LIN {X 0,Y 509.214,Z 871.751,A -85,B 0,C 180,E1 -5495.544,E2 -5495.544} C_VEL
LIN {X 0,Y 509.315,Z 866.896,A -85,B 0,C 180,E1 -5497.532,E2 -5497.532} C_VEL
LIN {X 0,Y 509.382,Z 861.752,A -85,B 0,C 180,E1 -5499.129,E2 -5499.129} C_VEL
LIN {X 0,Y 509.592,Z 855.435,A -85,B 0,C 180,E1 -5500.73,E2 -5500.73} C_VEL
LIN {X 0,Y 509.89,Z 847.858,A -85,B 0,C 180,E1 -5502.336,E2 -5502.336} C_VEL
LIN {X 0,Y 510.189,Z 840.077,A -85,B 0,C 180,E1 -5503.746,E2 -5503.746} C_VEL
LIN {X 0,Y 510.685,Z 831.046,A -85,B 0,C 180,E1 -5505.157,E2 -5505.157} C_VEL
LIN {X 0,Y 511.176,Z 820.613,A -85,B 0,C 180,E1 -5506.575,E2 -5506.575} C_VEL
LIN {X 0,Y 511.842,Z 808.389,A -85,B 0,C 180,E1 -5507.995,E2 -5507.995} C_VEL
LIN {X 0,Y 512.559,Z 796.031,A -85,B 0,C 180,E1 -5509.212,E2 -5509.212} C_VEL
LIN {X 0,Y 513.225,Z 784.136,A -85,B 0,C 180,E1 -5510.228,E2 -5510.228} C_VEL
LIN {X 0,Y 513.912,Z 772.243,A -85,B 0,C 180,E1 -5511.108,E2 -5511.108} C_VEL
LIN {X 0,Y 514.522,Z 760.984,A -85,B 0,C 180,E1 -5511.831,E2 -5511.831} C_VEL
LIN {X 0,Y 515.084,Z 748.665,A -85,B 0,C 180,E1 -5512.513,E2 -5512.513} C_VEL
LIN {X 0,Y 515.68,Z 735.496,A -85,B 0,C 180,E1 -5513.12,E2 -5513.12} C_VEL
LIN {X 0,Y 516.156,Z 722.774,A -85,B 0,C 180,E1 -5513.602,E2 -5513.602} C_VEL
LIN {X 0,Y 516.519,Z 710.205,A -85,B 0,C 180,E1 -5513.984,E2 -5513.984} C_VEL
LIN {X 0,Y 516.865,Z 696.063,A -85,B 0,C 180,E1 -5514.301,E2 -5514.301} C_VEL
LIN {X 0,Y 517.478,Z 641.628,A -85,B 0,C 180,E1 -5515.113,E2 -5515.113} C_VEL
LIN {X 0,Y 518.755,Z 504.01,A -85,B 0,C 180,E1 -5517.123,E2 -5517.123} C_VEL
LIN {X 0,Y 513.714,Z 483.814,A -85,B 0,C 180,E1 -5517.747,E2 -5517.747} C_VEL
LIN {X 0,Y 514.557,Z 463.773,A -85,B 0,C 180,E1 -5520.63,E2 -5520.63} C_VEL
LIN {X 0,Y 513.302,Z 457.477,A -85,B 0,C 180,E1 -5521.652,E2 -5521.652} C_VEL
LIN {X 0,Y 509.894,Z 444.343,A -85,B 0,C 180,E1 -5523.932,E2 -5523.932} C_VEL
LIN {X 0,Y 509.819,Z 444.213,A -85,B 0,C 180,E1 -5526.913,E2 -5526.913} C_VEL
LIN {X 0,Y 509.829,Z 444.217,A -85,B 0,C 180,E1 -5529.47,E2 -5529.47} C_VEL
LIN {X 0,Y 509.828,Z 444.222,A -85,B 0,C 180,E1 -5532.489,E2 -5532.489} C_VEL
LIN {X 0,Y 509.851,Z 444.222,A -85,B 0,C 180,E1 -5535.332,E2 -5535.332} C_VEL
LIN {X 0,Y 509.859,Z 444.219,A -85,B 0,C 180,E1 -5538.575,E2 -5538.575} C_VEL
LIN {X 0,Y 509.846,Z 444.227,A -85,B 0,C 180,E1 -5541.786,E2 -5541.786} C_VEL
LIN {X 0,Y 509.839,Z 444.212,A -85,B 0,C 180,E1 -5544.623,E2 -5544.623} C_VEL
LIN {X 0,Y 509.858,Z 444.222,A -85,B 0,C 180,E1 -5547.481,E2 -5547.481} C_VEL
LIN {X 0,Y 509.873,Z 444.209,A -85,B 0,C 180,E1 -5550.269,E2 -5550.269} C_VEL
LIN {X 0,Y 509.879,Z 444.208,A -85,B 0,C 180,E1 -5552.944,E2 -5552.944} C_VEL
LIN {X 0,Y 509.861,Z 444.222,A -85,B 0,C 180,E1 -5555.574,E2 -5555.574} C_VEL
LIN {X 0,Y 509.842,Z 444.205,A -85,B 0,C 180,E1 -5558.998,E2 -5558.998} C_VEL
LIN {X 0,Y 509.879,Z 444.21,A -85,B 0,C 180,E1 -5561.999,E2 -5561.999} C_VEL
LIN {X 0,Y 509.901,Z 444.215,A -85,B 0,C 180,E1 -5564.818,E2 -5564.818} C_VEL
LIN {X 0,Y 509.896,Z 444.218,A -85,B 0,C 180,E1 -5568.121,E2 -5568.121} C_VEL
LIN {X 0,Y 509.909,Z 444.207,A -85,B 0,C 180,E1 -5571.28,E2 -5571.28} C_VEL
LIN {X 0,Y 509.969,Z 444.207,A -85,B 0,C 180,E1 -5573.67,E2 -5573.67} C_VEL
LIN {X 0,Y 510.046,Z 444.194,A -85,B 0,C 180,E1 -5577.631,E2 -5577.631} C_VEL
LIN {X 0,Y 510.056,Z 444.192,A -85,B 0,C 180,E1 -5580.789,E2 -5580.789} C_VEL
LIN {X 0,Y 509.95,Z 444.209,A -85,B 0,C 180,E1 -5583.16,E2 -5583.16} C_VEL
LIN {X 0,Y 509.973,Z 444.205,A -85,B 0,C 180,E1 -5586.329,E2 -5586.329} C_VEL
LIN {X 0,Y 509.909,Z 444.22,A -85,B 0,C 180,E1 -5588.72,E2 -5588.72} C_VEL
LIN {X 0,Y 509.895,Z 444.211,A -85,B 0,C 180,E1 -5591.932,E2 -5591.932} C_VEL
LIN {X 0,Y 509.883,Z 444.213,A -85,B 0,C 180,E1 -5595.242,E2 -5595.242} C_VEL
LIN {X 0,Y 509.879,Z 444.218,A -85,B 0,C 180,E1 -5598.001,E2 -5598.001} C_VEL
LIN {X 0,Y 509.841,Z 444.226,A -85,B 0,C 180,E1 -5601.002,E2 -5601.002} C_VEL
LIN {X 0,Y 509.827,Z 444.223,A -85,B 0,C 180,E1 -5603.563,E2 -5603.563} C_VEL
LIN {X 0,Y 509.904,Z 444.2,A -85,B 0,C 180,E1 -5606.379,E2 -5606.379} C_VEL
LIN {X 0,Y 509.876,Z 444.216,A -85,B 0,C 180,E1 -5608.844,E2 -5608.844} C_VEL
LIN {X 0,Y 509.817,Z 444.224,A -85,B 0,C 180,E1 -5611.59,E2 -5611.59} C_VEL
LIN {X 0,Y 509.844,Z 444.204,A -85,B 0,C 180,E1 -5614.413,E2 -5614.413} C_VEL
LIN {X 0,Y 509.814,Z 444.233,A -85,B 0,C 180,E1 -5617.341,E2 -5617.341} C_VEL
LIN {X 0,Y 509.855,Z 444.222,A -85,B 0,C 180,E1 -5620.38,E2 -5620.38} C_VEL
LIN {X 0,Y 509.833,Z 444.231,A -85,B 0,C 180,E1 -5623.065,E2 -5623.065} C_VEL
LIN {X 0,Y 509.823,Z 444.228,A -85,B 0,C 180,E1 -5625.793,E2 -5625.793} C_VEL
LIN {X 0,Y 509.858,Z 444.222,A -85,B 0,C 180,E1 -5628.576,E2 -5628.576} C_VEL
LIN {X 0,Y 509.845,Z 444.227,A -85,B 0,C 180,E1 -5631.787,E2 -5631.787} C_VEL
LIN {X 0,Y 509.825,Z 444.229,A -85,B 0,C 180,E1 -5633.747,E2 -5633.747} C_VEL
LIN {X 0,Y 509.16,Z 444.309,A -85,B 0,C 180,E1 -5634.407,E2 -5634.407} C_VEL
LIN {X 0,Y 506.342,Z 444.666,A -85,B 0,C 180,E1 -5635.479,E2 -5635.479} C_VEL
LIN {X 0,Y 503.948,Z 444.964,A -85,B 0,C 180,E1 -5636.342,E2 -5636.342} C_VEL
LIN {X 0,Y 502.9,Z 445.092,A -85,B 0,C 180,E1 -5637.008,E2 -5637.008} C_VEL
LIN {X 0,Y 502.803,Z 445.102,A -85,B 0,C 180,E1 -5637.234,E2 -5637.234} C_VEL
LIN {X 0,Y 502.809,Z 445.102,A -85,B 0,C 180,E1 -5640.065,E2 -5640.065} C_VEL
LIN {X 0,Y 502.83,Z 445.097,A -85,B 0,C 180,E1 -5642.534,E2 -5642.534} C_VEL
LIN {X 0,Y 502.824,Z 445.103,A -85,B 0,C 180,E1 -5645.299,E2 -5645.299} C_VEL
LIN {X 0,Y 502.78,Z 445.109,A -85,B 0,C 180,E1 -5647.827,E2 -5647.827} C_VEL
LIN {X 0,Y 502.821,Z 445.1,A -85,B 0,C 180,E1 -5650.401,E2 -5650.401} C_VEL
LIN {X 0,Y 502.831,Z 445.097,A -85,B 0,C 180,E1 -5652.932,E2 -5652.932} C_VEL
LIN {X 0,Y 502.842,Z 445.101,A -85,B 0,C 180,E1 -5655.429,E2 -5655.429} C_VEL
LIN {X 0,Y 502.889,Z 445.091,A -85,B 0,C 180,E1 -5658.717,E2 -5658.717} C_VEL
LIN {X 0,Y 502.898,Z 445.094,A -85,B 0,C 180,E1 -5661.967,E2 -5661.967} C_VEL
LIN {X 0,Y 502.934,Z 445.088,A -85,B 0,C 180,E1 -5664.387,E2 -5664.387} C_VEL
LIN {X 0,Y 503.022,Z 445.078,A -85,B 0,C 180,E1 -5667.598,E2 -5667.598} C_VEL
LIN {X 0,Y 503.024,Z 445.08,A -85,B 0,C 180,E1 -5670,E2 -5670} C_VEL
LIN {X 0,Y 503.022,Z 445.078,A -85,B 0,C 180,E1 -5672.402,E2 -5672.402} C_VEL
LIN {X 0,Y 502.934,Z 445.087,A -85,B 0,C 180,E1 -5675.613,E2 -5675.613} C_VEL
LIN {X 0,Y 502.898,Z 445.094,A -85,B 0,C 180,E1 -5678.033,E2 -5678.033} C_VEL
LIN {X 0,Y 502.889,Z 445.091,A -85,B 0,C 180,E1 -5681.283,E2 -5681.283} C_VEL
LIN {X 0,Y 502.842,Z 445.101,A -85,B 0,C 180,E1 -5684.571,E2 -5684.571} C_VEL
LIN {X 0,Y 502.858,Z 445.097,A -85,B 0,C 180,E1 -5687.907,E2 -5687.907} C_VEL
LIN {X 0,Y 502.824,Z 445.104,A -85,B 0,C 180,E1 -5690.536,E2 -5690.536} C_VEL
LIN {X 0,Y 502.786,Z 445.105,A -85,B 0,C 180,E1 -5693.04,E2 -5693.04} C_VEL
LIN {X 0,Y 502.836,Z 445.097,A -85,B 0,C 180,E1 -5695.675,E2 -5695.675} C_VEL
LIN {X 0,Y 502.835,Z 445.102,A -85,B 0,C 180,E1 -5698.372,E2 -5698.372} C_VEL
LIN {X 0,Y 502.79,Z 445.102,A -85,B 0,C 180,E1 -5701.499,E2 -5701.499} C_VEL
LIN {X 0,Y 502.801,Z 445.106,A -85,B 0,C 180,E1 -5704.444,E2 -5704.444} C_VEL
LIN {X 0,Y 502.774,Z 445.106,A -85,B 0,C 180,E1 -5707.178,E2 -5707.178} C_VEL
LIN {X 0,Y 502.815,Z 445.1,A -85,B 0,C 180,E1 -5710.011,E2 -5710.011} C_VEL
LIN {X 0,Y 502.766,Z 445.108,A -85,B 0,C 180,E1 -5713.231,E2 -5713.231} C_VEL
LIN {X 0,Y 502.782,Z 445.103,A -85,B 0,C 180,E1 -5715.661,E2 -5715.661} C_VEL
LIN {X 0,Y 502.831,Z 445.097,A -85,B 0,C 180,E1 -5717.865,E2 -5717.865} C_VEL
LIN {X 0,Y 502.814,Z 445.105,A -85,B 0,C 180,E1 -5721.026,E2 -5721.026} C_VEL
LIN {X 0,Y 502.777,Z 445.101,A -85,B 0,C 180,E1 -5724.167,E2 -5724.167} C_VEL
LIN {X 0,Y 502.824,Z 445.086,A -85,B 0,C 180,E1 -5726.993,E2 -5726.993} C_VEL
LIN {X 0,Y 502.821,Z 445.097,A -85,B 0,C 180,E1 -5730.061,E2 -5730.061} C_VEL
LIN {X 0,Y 502.826,Z 445.085,A -85,B 0,C 180,E1 -5732.533,E2 -5732.533} C_VEL
LIN {X 0,Y 502.819,Z 445.095,A -85,B 0,C 180,E1 -5735.298,E2 -5735.298} C_VEL
LIN {X 0,Y 502.784,Z 445.102,A -85,B 0,C 180,E1 -5737.827,E2 -5737.827} C_VEL
LIN {X 0,Y 502.816,Z 445.094,A -85,B 0,C 180,E1 -5740.4,E2 -5740.4} C_VEL
LIN {X 0,Y 502.826,Z 445.101,A -85,B 0,C 180,E1 -5742.932,E2 -5742.932} C_VEL
LIN {X 0,Y 502.841,Z 445.1,A -85,B 0,C 180,E1 -5745.429,E2 -5745.429} C_VEL
LIN {X 0,Y 502.872,Z 445.086,A -85,B 0,C 180,E1 -5748.717,E2 -5748.717} C_VEL
LIN {X 0,Y 502.893,Z 445.087,A -85,B 0,C 180,E1 -5751.967,E2 -5751.967} C_VEL
LIN {X 0,Y 502.941,Z 445.078,A -85,B 0,C 180,E1 -5754.387,E2 -5754.387} C_VEL
LIN {X 0,Y 503.016,Z 445.072,A -85,B 0,C 180,E1 -5757.598,E2 -5757.598} C_VEL
LIN {X 0,Y 503.017,Z 445.075,A -85,B 0,C 180,E1 -5760,E2 -5760} C_VEL
LIN {X 0,Y 503.016,Z 445.07,A -85,B 0,C 180,E1 -5762.402,E2 -5762.402} C_VEL
LIN {X 0,Y 502.93,Z 445.09,A -85,B 0,C 180,E1 -5765.614,E2 -5765.614} C_VEL
LIN {X 0,Y 502.893,Z 445.083,A -85,B 0,C 180,E1 -5768.034,E2 -5768.034} C_VEL
LIN {X 0,Y 502.872,Z 445.093,A -85,B 0,C 180,E1 -5771.283,E2 -5771.283} C_VEL
LIN {X 0,Y 502.836,Z 445.094,A -85,B 0,C 180,E1 -5774.571,E2 -5774.571} C_VEL
LIN {X 0,Y 502.853,Z 445.086,A -85,B 0,C 180,E1 -5777.907,E2 -5777.907} C_VEL
LIN {X 0,Y 502.82,Z 445.078,A -85,B 0,C 180,E1 -5780.537,E2 -5780.537} C_VEL
LIN {X 0,Y 502.785,Z 445.099,A -85,B 0,C 180,E1 -5783.041,E2 -5783.041} C_VEL
LIN {X 0,Y 502.833,Z 445.101,A -85,B 0,C 180,E1 -5785.676,E2 -5785.676} C_VEL
LIN {X 0,Y 502.833,Z 445.079,A -85,B 0,C 180,E1 -5788.373,E2 -5788.373} C_VEL
LIN {X 0,Y 502.79,Z 445.102,A -85,B 0,C 180,E1 -5791.5,E2 -5791.5} C_VEL
LIN {X 0,Y 502.798,Z 445.09,A -85,B 0,C 180,E1 -5794.445,E2 -5794.445} C_VEL
LIN {X 0,Y 502.775,Z 445.103,A -85,B 0,C 180,E1 -5797.179,E2 -5797.179} C_VEL
LIN {X 0,Y 502.815,Z 445.094,A -85,B 0,C 180,E1 -5800.012,E2 -5800.012} C_VEL
LIN {X 0,Y 502.817,Z 445.106,A -85,B 0,C 180,E1 -5802.202,E2 -5802.202} C_VEL
LIN {X 0,Y 502.795,Z 445.101,A -85,B 0,C 180,E1 -5805.469,E2 -5805.469} C_VEL
LIN {X 0,Y 502.816,Z 445.103,A -85,B 0,C 180,E1 -5808.935,E2 -5808.935} C_VEL
LIN {X 0,Y 502.789,Z 445.077,A -85,B 0,C 180,E1 -5812.047,E2 -5812.047} C_VEL
LIN {X 0,Y 502.806,Z 445.09,A -85,B 0,C 180,E1 -5815.036,E2 -5815.036} C_VEL
LIN {X 0,Y 502.864,Z 445.312,A -85,B 0,C 180,E1 -5815.728,E2 -5815.728} C_VEL
LIN {X 0,Y 506.903,Z 460.784,A -85,B 0,C 180,E1 -5818.441,E2 -5818.441} C_VEL
LIN {X 0,Y 507.802,Z 465.396,A -85,B 0,C 180,E1 -5819.198,E2 -5819.198} C_VEL
LIN {X 0,Y 507.008,Z 483.571,A -85,B 0,C 180,E1 -5821.854,E2 -5821.854} C_VEL
LIN {X 0,Y 512.435,Z 505.265,A -85,B 0,C 180,E1 -5822.537,E2 -5822.537} C_VEL
LIN {X 0,Y 510.952,Z 650.451,A -85,B 0,C 180,E1 -5824.68,E2 -5824.68} C_VEL
LIN {X 0,Y 510.401,Z 694.978,A -85,B 0,C 180,E1 -5825.352,E2 -5825.352} C_VEL
LIN {X 0,Y 510.117,Z 707.15,A -85,B 0,C 180,E1 -5825.614,E2 -5825.614} C_VEL
LIN {X 0,Y 509.708,Z 720.461,A -85,B 0,C 180,E1 -5825.999,E2 -5825.999} C_VEL
LIN {X 0,Y 509.225,Z 733.017,A -85,B 0,C 180,E1 -5826.461,E2 -5826.461} C_VEL
LIN {X 0,Y 508.632,Z 745.582,A -85,B 0,C 180,E1 -5827.025,E2 -5827.025} C_VEL
LIN {X 0,Y 508.086,Z 757.162,A -85,B 0,C 180,E1 -5827.643,E2 -5827.643} C_VEL
LIN {X 0,Y 507.441,Z 768.687,A -85,B 0,C 180,E1 -5828.357,E2 -5828.357} C_VEL
LIN {X 0,Y 506.627,Z 781.53,A -85,B 0,C 180,E1 -5829.284,E2 -5829.284} C_VEL
LIN {X 0,Y 505.986,Z 792.61,A -85,B 0,C 180,E1 -5830.211,E2 -5830.211} C_VEL
LIN {X 0,Y 505.371,Z 802.694,A -85,B 0,C 180,E1 -5831.168,E2 -5831.168} C_VEL
LIN {X 0,Y 504.77,Z 812.019,A -85,B 0,C 180,E1 -5832.163,E2 -5832.163} C_VEL
LIN {X 0,Y 504.146,Z 822.161,A -85,B 0,C 180,E1 -5833.395,E2 -5833.395} C_VEL
LIN {X 0,Y 503.707,Z 831.043,A -85,B 0,C 180,E1 -5834.628,E2 -5834.628} C_VEL
LIN {X 0,Y 503.261,Z 838.873,A -85,B 0,C 180,E1 -5835.855,E2 -5835.855} C_VEL
LIN {X 0,Y 502.915,Z 846.81,A -85,B 0,C 180,E1 -5837.285,E2 -5837.285} C_VEL
LIN {X 0,Y 502.737,Z 851.639,A -85,B 0,C 180,E1 -5838.26,E2 -5838.26} C_VEL
LIN {X 0,Y 502.417,Z 858.713,A -85,B 0,C 180,E1 -5839.93,E2 -5839.93} C_VEL
LIN {X 0,Y 502.272,Z 864.389,A -85,B 0,C 180,E1 -5841.552,E2 -5841.552} C_VEL
LIN {X 0,Y 502.23,Z 867.952,A -85,B 0,C 180,E1 -5842.765,E2 -5842.765} C_VEL
LIN {X 0,Y 502.131,Z 871.746,A -85,B 0,C 180,E1 -5844.378,E2 -5844.378} C_VEL
LIN {X 0,Y 502.088,Z 874.537,A -85,B 0,C 180,E1 -5845.987,E2 -5845.987} C_VEL
LIN {X 0,Y 502.058,Z 876.394,A -85,B 0,C 180,E1 -5847.593,E2 -5847.593} C_VEL
LIN {X 0,Y 501.985,Z 877.31,A -85,B 0,C 180,E1 -5849.198,E2 -5849.198} C_VEL
LIN {X 0,Y 501.985,Z 877.31,A -85,B 0,C 180,E1 -5850.802,E2 -5850.802} C_VEL
LIN {X 0,Y 502.058,Z 876.394,A -85,B 0,C 180,E1 -5852.407,E2 -5852.407} C_VEL
LIN {X 0,Y 502.088,Z 874.537,A -85,B 0,C 180,E1 -5854.013,E2 -5854.013} C_VEL
LIN {X 0,Y 502.131,Z 871.746,A -85,B 0,C 180,E1 -5855.622,E2 -5855.622} C_VEL
LIN {X 0,Y 502.23,Z 867.952,A -85,B 0,C 180,E1 -5857.235,E2 -5857.235} C_VEL
LIN {X 0,Y 502.322,Z 861.755,A -85,B 0,C 180,E1 -5859.259,E2 -5859.259} C_VEL
LIN {X 0,Y 502.55,Z 855.432,A -85,B 0,C 180,E1 -5860.882,E2 -5860.882} C_VEL
LIN {X 0,Y 502.817,Z 848.895,A -85,B 0,C 180,E1 -5862.307,E2 -5862.307} C_VEL
LIN {X 0,Y 503.138,Z 841.269,A -85,B 0,C 180,E1 -5863.736,E2 -5863.736} C_VEL
LIN {X 0,Y 503.585,Z 833.778,A -85,B 0,C 180,E1 -5864.962,E2 -5864.962} C_VEL
LIN {X 0,Y 504.015,Z 825.271,A -85,B 0,C 180,E1 -5866.193,E2 -5866.193} C_VEL
LIN {X 0,Y 504.551,Z 815.547,A -85,B 0,C 180,E1 -5867.426,E2 -5867.426} C_VEL
LIN {X 0,Y 505.264,Z 804.394,A -85,B 0,C 180,E1 -5868.658,E2 -5868.658} C_VEL
LIN {X 0,Y 505.915,Z 793.748,A -85,B 0,C 180,E1 -5869.686,E2 -5869.686} C_VEL
LIN {X 0,Y 506.55,Z 782.829,A -85,B 0,C 180,E1 -5870.613,E2 -5870.613} C_VEL
LIN {X 0,Y 507.29,Z 771.289,A -85,B 0,C 180,E1 -5871.464,E2 -5871.464} C_VEL
LIN {X 0,Y 507.927,Z 760.627,A -85,B 0,C 180,E1 -5872.15,E2 -5872.15} C_VEL
LIN {X 0,Y 508.508,Z 748.652,A -85,B 0,C 180,E1 -5872.82,E2 -5872.82} C_VEL
LIN {X 0,Y 509.08,Z 736.712,A -85,B 0,C 180,E1 -5873.384,E2 -5873.384} C_VEL
LIN {X 0,Y 509.623,Z 723.528,A -85,B 0,C 180,E1 -5873.897,E2 -5873.897} C_VEL
LIN {X 0,Y 510.043,Z 710.15,A -85,B 0,C 180,E1 -5874.308,E2 -5874.308} C_VEL
LIN {X 0,Y 510.392,Z 697.165,A -85,B 0,C 180,E1 -5874.606,E2 -5874.606} C_VEL
LIN {X 0,Y 510.808,Z 662.532,A -85,B 0,C 180,E1 -5875.144,E2 -5875.144} C_VEL
LIN {X 0,Y 512.439,Z 505.381,A -85,B 0,C 180,E1 -5877.461,E2 -5877.461} C_VEL
LIN {X 0,Y 507.014,Z 483.552,A -85,B 0,C 180,E1 -5878.146,E2 -5878.146} C_VEL
LIN {X 0,Y 507.798,Z 465.396,A -85,B 0,C 180,E1 -5880.802,E2 -5880.802} C_VEL
LIN {X 0,Y 506.049,Z 457.64,A -85,B 0,C 180,E1 -5882.095,E2 -5882.095} C_VEL
LIN {X 0,Y 502.864,Z 445.298,A -85,B 0,C 180,E1 -5884.272,E2 -5884.272} C_VEL
LIN {X 0,Y 502.773,Z 445.088,A -85,B 0,C 180,E1 -5886.946,E2 -5886.946} C_VEL
LIN {X 0,Y 502.783,Z 445.105,A -85,B 0,C 180,E1 -5890.015,E2 -5890.015} C_VEL
LIN {X 0,Y 502.797,Z 445.098,A -85,B 0,C 180,E1 -5892.199,E2 -5892.199} C_VEL
LIN {X 0,Y 502.795,Z 445.099,A -85,B 0,C 180,E1 -5895.468,E2 -5895.468} C_VEL
LIN {X 0,Y 502.829,Z 445.103,A -85,B 0,C 180,E1 -5897.864,E2 -5897.864} C_VEL
LIN {X 0,Y 502.803,Z 445.095,A -85,B 0,C 180,E1 -5901.024,E2 -5901.024} C_VEL
LIN {X 0,Y 502.779,Z 445.095,A -85,B 0,C 180,E1 -5904.167,E2 -5904.167} C_VEL
LIN {X 0,Y 502.825,Z 445.095,A -85,B 0,C 180,E1 -5906.993,E2 -5906.993} C_VEL
LIN {X 0,Y 502.822,Z 445.09,A -85,B 0,C 180,E1 -5910.061,E2 -5910.061} C_VEL
LIN {X 0,Y 502.827,Z 445.086,A -85,B 0,C 180,E1 -5912.533,E2 -5912.533} C_VEL
LIN {X 0,Y 502.82,Z 445.097,A -85,B 0,C 180,E1 -5915.298,E2 -5915.298} C_VEL
LIN {X 0,Y 502.772,Z 445.1,A -85,B 0,C 180,E1 -5917.826,E2 -5917.826} C_VEL
LIN {X 0,Y 502.816,Z 445.079,A -85,B 0,C 180,E1 -5920.4,E2 -5920.4} C_VEL
LIN {X 0,Y 502.827,Z 445.094,A -85,B 0,C 180,E1 -5922.931,E2 -5922.931} C_VEL
LIN {X 0,Y 502.836,Z 445.094,A -85,B 0,C 180,E1 -5925.429,E2 -5925.429} C_VEL
LIN {X 0,Y 502.872,Z 445.093,A -85,B 0,C 180,E1 -5928.717,E2 -5928.717} C_VEL
LIN {X 0,Y 502.893,Z 445.084,A -85,B 0,C 180,E1 -5931.966,E2 -5931.966} C_VEL
LIN {X 0,Y 502.93,Z 445.091,A -85,B 0,C 180,E1 -5934.386,E2 -5934.386} C_VEL
LIN {X 0,Y 503.016,Z 445.07,A -85,B 0,C 180,E1 -5937.598,E2 -5937.598} C_VEL
LIN {X 0,Y 503.017,Z 445.074,A -85,B 0,C 180,E1 -5940,E2 -5940} C_VEL
LIN {X 0,Y 503.016,Z 445.071,A -85,B 0,C 180,E1 -5942.402,E2 -5942.402} C_VEL
LIN {X 0,Y 502.941,Z 445.077,A -85,B 0,C 180,E1 -5945.613,E2 -5945.613} C_VEL
LIN {X 0,Y 502.893,Z 445.086,A -85,B 0,C 180,E1 -5948.033,E2 -5948.033} C_VEL
LIN {X 0,Y 502.872,Z 445.086,A -85,B 0,C 180,E1 -5951.283,E2 -5951.283} C_VEL
LIN {X 0,Y 502.841,Z 445.1,A -85,B 0,C 180,E1 -5954.571,E2 -5954.571} C_VEL
LIN {X 0,Y 502.852,Z 445.093,A -85,B 0,C 180,E1 -5957.907,E2 -5957.907} C_VEL
LIN {X 0,Y 502.819,Z 445.097,A -85,B 0,C 180,E1 -5960.536,E2 -5960.536} C_VEL
LIN {X 0,Y 502.787,Z 445.106,A -85,B 0,C 180,E1 -5963.04,E2 -5963.04} C_VEL
LIN {X 0,Y 502.832,Z 445.079,A -85,B 0,C 180,E1 -5965.676,E2 -5965.676} C_VEL
LIN {X 0,Y 502.833,Z 445.087,A -85,B 0,C 180,E1 -5968.373,E2 -5968.373} C_VEL
LIN {X 0,Y 502.788,Z 445.101,A -85,B 0,C 180,E1 -5971.5,E2 -5971.5} C_VEL
LIN {X 0,Y 502.797,Z 445.081,A -85,B 0,C 180,E1 -5974.445,E2 -5974.445} C_VEL
LIN {X 0,Y 502.775,Z 445.111,A -85,B 0,C 180,E1 -5977.179,E2 -5977.179} C_VEL
LIN {X 0,Y 502.819,Z 445.098,A -85,B 0,C 180,E1 -5980.012,E2 -5980.012} C_VEL
LIN {X 0,Y 502.818,Z 445.098,A -85,B 0,C 180,E1 -5982.203,E2 -5982.203} C_VEL
LIN {X 0,Y 502.793,Z 445.107,A -85,B 0,C 180,E1 -5985.469,E2 -5985.469} C_VEL
LIN {X 0,Y 502.819,Z 445.102,A -85,B 0,C 180,E1 -5989.004,E2 -5989.004} C_VEL
LIN {X 0,Y 502.788,Z 445.104,A -85,B 0,C 180,E1 -5992.047,E2 -5992.047} C_VEL
LIN {X 0,Y 502.804,Z 445.103,A -85,B 0,C 180,E1 -5995.036,E2 -5995.036} C_VEL
LIN {X 0,Y 502.803,Z 445.102,A -85,B 0,C 180,E1 -5997.234,E2 -5997.234} C_VEL
LIN {X 0,Y 502.103,Z 445.191,A -85,B 0,C 180,E1 -5997.903,E2 -5997.903} C_VEL
LIN {X 0,Y 499.238,Z 445.547,A -85,B 0,C 180,E1 -5998.988,E2 -5998.988} C_VEL
LIN {X 0,Y 496.842,Z 445.847,A -85,B 0,C 180,E1 -5999.863,E2 -5999.863} C_VEL
LIN {X 0,Y 495.825,Z 445.97,A -85,B 0,C 180,E1 -6000.539,E2 -6000.539} C_VEL
LIN {X 0,Y 495.748,Z 445.98,A -85,B 0,C 180,E1 -6000.768,E2 -6000.768} C_VEL
LIN {X 0,Y 495.795,Z 445.977,A -85,B 0,C 180,E1 -6003.933,E2 -6003.933} C_VEL
LIN {X 0,Y 495.761,Z 445.981,A -85,B 0,C 180,E1 -6007.138,E2 -6007.138} C_VEL
LIN {X 0,Y 495.768,Z 445.981,A -85,B 0,C 180,E1 -6010.11,E2 -6010.11} C_VEL
LIN {X 0,Y 495.783,Z 445.975,A -85,B 0,C 180,E1 -6012.682,E2 -6012.682} C_VEL
LIN {X 0,Y 495.786,Z 445.978,A -85,B 0,C 180,E1 -6015.217,E2 -6015.217} C_VEL
LIN {X 0,Y 495.864,Z 445.967,A -85,B 0,C 180,E1 -6018.555,E2 -6018.555} C_VEL
LIN {X 0,Y 495.869,Z 445.971,A -85,B 0,C 180,E1 -6021.852,E2 -6021.852} C_VEL
LIN {X 0,Y 495.892,Z 445.966,A -85,B 0,C 180,E1 -6024.307,E2 -6024.307} C_VEL
LIN {X 0,Y 495.991,Z 445.954,A -85,B 0,C 180,E1 -6027.564,E2 -6027.564} C_VEL
LIN {X 0,Y 495.996,Z 445.956,A -85,B 0,C 180,E1 -6030,E2 -6030} C_VEL
LIN {X 0,Y 495.991,Z 445.954,A -85,B 0,C 180,E1 -6032.436,E2 -6032.436} C_VEL
LIN {X 0,Y 495.892,Z 445.966,A -85,B 0,C 180,E1 -6035.693,E2 -6035.693} C_VEL
LIN {X 0,Y 495.869,Z 445.971,A -85,B 0,C 180,E1 -6038.148,E2 -6038.148} C_VEL
LIN {X 0,Y 495.864,Z 445.967,A -85,B 0,C 180,E1 -6041.445,E2 -6041.445} C_VEL
LIN {X 0,Y 495.786,Z 445.978,A -85,B 0,C 180,E1 -6044.783,E2 -6044.783} C_VEL
LIN {X 0,Y 495.784,Z 445.974,A -85,B 0,C 180,E1 -6047.318,E2 -6047.318} C_VEL
LIN {X 0,Y 495.768,Z 445.981,A -85,B 0,C 180,E1 -6049.89,E2 -6049.89} C_VEL
LIN {X 0,Y 495.755,Z 445.982,A -85,B 0,C 180,E1 -6052.86,E2 -6052.86} C_VEL
LIN {X 0,Y 495.794,Z 445.977,A -85,B 0,C 180,E1 -6056.067,E2 -6056.067} C_VEL
LIN {X 0,Y 495.767,Z 445.982,A -85,B 0,C 180,E1 -6058.814,E2 -6058.814} C_VEL
LIN {X 0,Y 495.753,Z 445.979,A -85,B 0,C 180,E1 -6061.726,E2 -6061.726} C_VEL
LIN {X 0,Y 495.771,Z 445.983,A -85,B 0,C 180,E1 -6064.695,E2 -6064.695} C_VEL
LIN {X 0,Y 495.725,Z 445.983,A -85,B 0,C 180,E1 -6067.561,E2 -6067.561} C_VEL
LIN {X 0,Y 495.773,Z 445.983,A -85,B 0,C 180,E1 -6070.698,E2 -6070.698} C_VEL
LIN {X 0,Y 495.726,Z 445.983,A -85,B 0,C 180,E1 -6074.001,E2 -6074.001} C_VEL
LIN {X 0,Y 495.756,Z 445.983,A -85,B 0,C 180,E1 -6077.121,E2 -6077.121} C_VEL
LIN {X 0,Y 495.783,Z 445.977,A -85,B 0,C 180,E1 -6080.365,E2 -6080.365} C_VEL
LIN {X 0,Y 495.726,Z 445.98,A -85,B 0,C 180,E1 -6083.456,E2 -6083.456} C_VEL
LIN {X 0,Y 495.752,Z 445.958,A -85,B 0,C 180,E1 -6086.436,E2 -6086.436} C_VEL
LIN {X 0,Y 495.748,Z 445.983,A -85,B 0,C 180,E1 -6089.313,E2 -6089.313} C_VEL
LIN {X 0,Y 495.774,Z 445.964,A -85,B 0,C 180,E1 -6092.109,E2 -6092.109} C_VEL
LIN {X 0,Y 495.78,Z 445.962,A -85,B 0,C 180,E1 -6094.833,E2 -6094.833} C_VEL
LIN {X 0,Y 495.74,Z 445.983,A -85,B 0,C 180,E1 -6097.495,E2 -6097.495} C_VEL
LIN {X 0,Y 495.768,Z 445.972,A -85,B 0,C 180,E1 -6100.11,E2 -6100.11} C_VEL
LIN {X 0,Y 495.778,Z 445.976,A -85,B 0,C 180,E1 -6102.681,E2 -6102.681} C_VEL
LIN {X 0,Y 495.784,Z 445.975,A -85,B 0,C 180,E1 -6105.217,E2 -6105.217} C_VEL
LIN {X 0,Y 495.845,Z 445.96,A -85,B 0,C 180,E1 -6108.555,E2 -6108.555} C_VEL
LIN {X 0,Y 495.864,Z 445.963,A -85,B 0,C 180,E1 -6111.852,E2 -6111.852} C_VEL
LIN {X 0,Y 495.897,Z 445.955,A -85,B 0,C 180,E1 -6114.307,E2 -6114.307} C_VEL
LIN {X 0,Y 495.984,Z 445.948,A -85,B 0,C 180,E1 -6117.564,E2 -6117.564} C_VEL
LIN {X 0,Y 495.988,Z 445.95,A -85,B 0,C 180,E1 -6120,E2 -6120} C_VEL
LIN {X 0,Y 495.985,Z 445.946,A -85,B 0,C 180,E1 -6122.436,E2 -6122.436} C_VEL
LIN {X 0,Y 495.887,Z 445.968,A -85,B 0,C 180,E1 -6125.694,E2 -6125.694} C_VEL
LIN {X 0,Y 495.864,Z 445.957,A -85,B 0,C 180,E1 -6128.148,E2 -6128.148} C_VEL
LIN {X 0,Y 495.846,Z 445.97,A -85,B 0,C 180,E1 -6131.445,E2 -6131.445} C_VEL
LIN {X 0,Y 495.781,Z 445.972,A -85,B 0,C 180,E1 -6134.783,E2 -6134.783} C_VEL
LIN {X 0,Y 495.779,Z 445.974,A -85,B 0,C 180,E1 -6137.319,E2 -6137.319} C_VEL
LIN {X 0,Y 495.762,Z 445.954,A -85,B 0,C 180,E1 -6139.891,E2 -6139.891} C_VEL
LIN {X 0,Y 495.753,Z 445.974,A -85,B 0,C 180,E1 -6142.862,E2 -6142.862} C_VEL
LIN {X 0,Y 495.791,Z 445.97,A -85,B 0,C 180,E1 -6146.068,E2 -6146.068} C_VEL
LIN {X 0,Y 495.771,Z 445.959,A -85,B 0,C 180,E1 -6148.815,E2 -6148.815} C_VEL
LIN {X 0,Y 495.752,Z 445.981,A -85,B 0,C 180,E1 -6151.727,E2 -6151.727} C_VEL
LIN {X 0,Y 495.769,Z 445.963,A -85,B 0,C 180,E1 -6154.696,E2 -6154.696} C_VEL
LIN {X 0,Y 495.725,Z 445.983,A -85,B 0,C 180,E1 -6157.562,E2 -6157.562} C_VEL
LIN {X 0,Y 495.773,Z 445.974,A -85,B 0,C 180,E1 -6160.699,E2 -6160.699} C_VEL
LIN {X 0,Y 495.728,Z 445.98,A -85,B 0,C 180,E1 -6163.696,E2 -6163.696} C_VEL
LIN {X 0,Y 495.723,Z 445.987,A -85,B 0,C 180,E1 -6166.306,E2 -6166.306} C_VEL
LIN {X 0,Y 495.762,Z 445.98,A -85,B 0,C 180,E1 -6169.301,E2 -6169.301} C_VEL
LIN {X 0,Y 495.726,Z 445.955,A -85,B 0,C 180,E1 -6172.439,E2 -6172.439} C_VEL
LIN {X 0,Y 495.774,Z 446.061,A -85,B 0,C 180,E1 -6175.305,E2 -6175.305} C_VEL
LIN {X 0,Y 497.409,Z 452.245,A -85,B 0,C 180,E1 -6176.473,E2 -6176.473} C_VEL
LIN {X 0,Y 500.903,Z 465.996,A -85,B 0,C 180,E1 -6178.856,E2 -6178.856} C_VEL
LIN {X 0,Y 500.878,Z 471.265,A -85,B 0,C 180,E1 -6179.661,E2 -6179.661} C_VEL
LIN {X 0,Y 500.294,Z 483.313,A -85,B 0,C 180,E1 -6181.442,E2 -6181.442} C_VEL
LIN {X 0,Y 506.144,Z 506.915,A -85,B 0,C 180,E1 -6182.195,E2 -6182.195} C_VEL
LIN {X 0,Y 504.265,Z 674.916,A -85,B 0,C 180,E1 -6184.701,E2 -6184.701} C_VEL
LIN {X 0,Y 503.854,Z 700.354,A -85,B 0,C 180,E1 -6185.118,E2 -6185.118} C_VEL
LIN {X 0,Y 503.311,Z 717.951,A -85,B 0,C 180,E1 -6185.593,E2 -6185.593} C_VEL
LIN {X 0,Y 502.705,Z 731.596,A -85,B 0,C 180,E1 -6186.082,E2 -6186.082} C_VEL
LIN {X 0,Y 502.129,Z 744.412,A -85,B 0,C 180,E1 -6186.655,E2 -6186.655} C_VEL
LIN {X 0,Y 501.452,Z 757.059,A -85,B 0,C 180,E1 -6187.331,E2 -6187.331} C_VEL
LIN {X 0,Y 500.744,Z 769.56,A -85,B 0,C 180,E1 -6188.119,E2 -6188.119} C_VEL
LIN {X 0,Y 499.916,Z 781.522,A -85,B 0,C 180,E1 -6188.993,E2 -6188.993} C_VEL
LIN {X 0,Y 499.252,Z 792.603,A -85,B 0,C 180,E1 -6189.933,E2 -6189.933} C_VEL
LIN {X 0,Y 498.507,Z 803.445,A -85,B 0,C 180,E1 -6190.98,E2 -6190.98} C_VEL
LIN {X 0,Y 497.817,Z 813.778,A -85,B 0,C 180,E1 -6192.118,E2 -6192.118} C_VEL
LIN {X 0,Y 497.241,Z 822.154,A -85,B 0,C 180,E1 -6193.158,E2 -6193.158} C_VEL
LIN {X 0,Y 496.753,Z 831.039,A -85,B 0,C 180,E1 -6194.407,E2 -6194.407} C_VEL
LIN {X 0,Y 496.287,Z 838.867,A -85,B 0,C 180,E1 -6195.652,E2 -6195.652} C_VEL
LIN {X 0,Y 495.893,Z 846.805,A -85,B 0,C 180,E1 -6197.102,E2 -6197.102} C_VEL
LIN {X 0,Y 495.584,Z 853.632,A -85,B 0,C 180,E1 -6198.549,E2 -6198.549} C_VEL
LIN {X 0,Y 495.366,Z 858.707,A -85,B 0,C 180,E1 -6199.785,E2 -6199.785} C_VEL
LIN {X 0,Y 495.183,Z 864.385,A -85,B 0,C 180,E1 -6201.43,E2 -6201.43} C_VEL
LIN {X 0,Y 495.149,Z 867.948,A -85,B 0,C 180,E1 -6202.661,E2 -6202.661} C_VEL
LIN {X 0,Y 495.052,Z 871.741,A -85,B 0,C 180,E1 -6204.297,E2 -6204.297} C_VEL
LIN {X 0,Y 494.984,Z 874.534,A -85,B 0,C 180,E1 -6205.929,E2 -6205.929} C_VEL
LIN {X 0,Y 495.023,Z 875.648,A -85,B 0,C 180,E1 -6206.745,E2 -6206.745} C_VEL
LIN {X 0,Y 494.955,Z 877.03,A -85,B 0,C 180,E1 -6208.373,E2 -6208.373} C_VEL
LIN {X 0,Y 494.893,Z 877.5,A -85,B 0,C 180,E1 -6210,E2 -6210} C_VEL
LIN {X 0,Y 494.955,Z 877.03,A -85,B 0,C 180,E1 -6211.627,E2 -6211.627} C_VEL
LIN {X 0,Y 495.023,Z 875.648,A -85,B 0,C 180,E1 -6213.255,E2 -6213.255} C_VEL
LIN {X 0,Y 494.982,Z 873.314,A -85,B 0,C 180,E1 -6214.887,E2 -6214.887} C_VEL
LIN {X 0,Y 495.112,Z 868.971,A -85,B 0,C 180,E1 -6216.93,E2 -6216.93} C_VEL
LIN {X 0,Y 495.176,Z 865.654,A -85,B 0,C 180,E1 -6218.159,E2 -6218.159} C_VEL
LIN {X 0,Y 495.271,Z 860.232,A -85,B 0,C 180,E1 -6219.804,E2 -6219.804} C_VEL
LIN {X 0,Y 495.501,Z 855.428,A -85,B 0,C 180,E1 -6221.039,E2 -6221.039} C_VEL
LIN {X 0,Y 495.851,Z 847.848,A -85,B 0,C 180,E1 -6222.691,E2 -6222.691} C_VEL
LIN {X 0,Y 496.233,Z 840.065,A -85,B 0,C 180,E1 -6224.141,E2 -6224.141} C_VEL
LIN {X 0,Y 496.708,Z 832.407,A -85,B 0,C 180,E1 -6225.384,E2 -6225.384} C_VEL
LIN {X 0,Y 497.186,Z 823.709,A -85,B 0,C 180,E1 -6226.633,E2 -6226.633} C_VEL
LIN {X 0,Y 497.688,Z 815.542,A -85,B 0,C 180,E1 -6227.674,E2 -6227.674} C_VEL
LIN {X 0,Y 498.445,Z 804.386,A -85,B 0,C 180,E1 -6228.923,E2 -6228.923} C_VEL
LIN {X 0,Y 499.157,Z 793.741,A -85,B 0,C 180,E1 -6229.964,E2 -6229.964} C_VEL
LIN {X 0,Y 499.823,Z 782.821,A -85,B 0,C 180,E1 -6230.903,E2 -6230.903} C_VEL
LIN {X 0,Y 500.598,Z 771.603,A -85,B 0,C 180,E1 -6231.74,E2 -6231.74} C_VEL
LIN {X 0,Y 501.276,Z 760.546,A -85,B 0,C 180,E1 -6232.46,E2 -6232.46} C_VEL
LIN {X 0,Y 501.921,Z 748.52,A -85,B 0,C 180,E1 -6233.137,E2 -6233.137} C_VEL
LIN {X 0,Y 502.53,Z 736.539,A -85,B 0,C 180,E1 -6233.707,E2 -6233.707} C_VEL
LIN {X 0,Y 503.103,Z 723.318,A -85,B 0,C 180,E1 -6234.226,E2 -6234.226} C_VEL
LIN {X 0,Y 503.568,Z 709.94,A -85,B 0,C 180,E1 -6234.641,E2 -6234.641} C_VEL
LIN {X 0,Y 503.941,Z 696.661,A -85,B 0,C 180,E1 -6234.949,E2 -6234.949} C_VEL
LIN {X 0,Y 504.434,Z 659.104,A -85,B 0,C 180,E1 -6235.534,E2 -6235.534} C_VEL
LIN {X 0,Y 506.161,Z 506.735,A -85,B 0,C 180,E1 -6237.806,E2 -6237.806} C_VEL
LIN {X 0,Y 500.329,Z 483.29,A -85,B 0,C 180,E1 -6238.556,E2 -6238.556} C_VEL
LIN {X 0,Y 501.056,Z 467.121,A -85,B 0,C 180,E1 -6240.962,E2 -6240.962} C_VEL
LIN {X 0,Y 498.356,Z 455.899,A -85,B 0,C 180,E1 -6242.883,E2 -6242.883} C_VEL
LIN {X 0,Y 495.835,Z 446.308,A -85,B 0,C 180,E1 -6244.616,E2 -6244.616} C_VEL
LIN {X 0,Y 495.764,Z 445.961,A -85,B 0,C 180,E1 -6244.849,E2 -6244.849} C_VEL
LIN {X 0,Y 495.726,Z 445.956,A -85,B 0,C 180,E1 -6247.561,E2 -6247.561} C_VEL
LIN {X 0,Y 495.761,Z 445.981,A -85,B 0,C 180,E1 -6250.699,E2 -6250.699} C_VEL
LIN {X 0,Y 495.728,Z 445.986,A -85,B 0,C 180,E1 -6254,E2 -6254} C_VEL
LIN {X 0,Y 495.757,Z 445.977,A -85,B 0,C 180,E1 -6257.12,E2 -6257.12} C_VEL
LIN {X 0,Y 495.777,Z 445.971,A -85,B 0,C 180,E1 -6260.364,E2 -6260.364} C_VEL
LIN {X 0,Y 495.728,Z 445.985,A -85,B 0,C 180,E1 -6263.456,E2 -6263.456} C_VEL
LIN {X 0,Y 495.753,Z 445.978,A -85,B 0,C 180,E1 -6266.435,E2 -6266.435} C_VEL
LIN {X 0,Y 495.75,Z 445.978,A -85,B 0,C 180,E1 -6269.313,E2 -6269.313} C_VEL
LIN {X 0,Y 495.774,Z 445.958,A -85,B 0,C 180,E1 -6272.108,E2 -6272.108} C_VEL
LIN {X 0,Y 495.781,Z 445.974,A -85,B 0,C 180,E1 -6274.832,E2 -6274.832} C_VEL
LIN {X 0,Y 495.741,Z 445.977,A -85,B 0,C 180,E1 -6277.494,E2 -6277.494} C_VEL
LIN {X 0,Y 495.762,Z 445.954,A -85,B 0,C 180,E1 -6280.109,E2 -6280.109} C_VEL
LIN {X 0,Y 495.779,Z 445.974,A -85,B 0,C 180,E1 -6282.681,E2 -6282.681} C_VEL
LIN {X 0,Y 495.781,Z 445.972,A -85,B 0,C 180,E1 -6285.217,E2 -6285.217} C_VEL
LIN {X 0,Y 495.846,Z 445.971,A -85,B 0,C 180,E1 -6288.555,E2 -6288.555} C_VEL
LIN {X 0,Y 495.864,Z 445.958,A -85,B 0,C 180,E1 -6291.852,E2 -6291.852} C_VEL
LIN {X 0,Y 495.887,Z 445.969,A -85,B 0,C 180,E1 -6294.306,E2 -6294.306} C_VEL
LIN {X 0,Y 495.985,Z 445.946,A -85,B 0,C 180,E1 -6297.564,E2 -6297.564} C_VEL
LIN {X 0,Y 495.988,Z 445.95,A -85,B 0,C 180,E1 -6300,E2 -6300} C_VEL
LIN {X 0,Y 495.984,Z 445.947,A -85,B 0,C 180,E1 -6302.436,E2 -6302.436} C_VEL
LIN {X 0,Y 495.897,Z 445.954,A -85,B 0,C 180,E1 -6305.693,E2 -6305.693} C_VEL
LIN {X 0,Y 495.864,Z 445.963,A -85,B 0,C 180,E1 -6308.148,E2 -6308.148} C_VEL
LIN {X 0,Y 495.845,Z 445.961,A -85,B 0,C 180,E1 -6311.445,E2 -6311.445} C_VEL
LIN {X 0,Y 495.784,Z 445.975,A -85,B 0,C 180,E1 -6314.783,E2 -6314.783} C_VEL
LIN {X 0,Y 495.778,Z 445.977,A -85,B 0,C 180,E1 -6317.319,E2 -6317.319} C_VEL
LIN {X 0,Y 495.768,Z 445.972,A -85,B 0,C 180,E1 -6319.89,E2 -6319.89} C_VEL
LIN {X 0,Y 495.748,Z 445.986,A -85,B 0,C 180,E1 -6322.86,E2 -6322.86} C_VEL
LIN {X 0,Y 495.79,Z 445.955,A -85,B 0,C 180,E1 -6326.068,E2 -6326.068} C_VEL
LIN {X 0,Y 495.771,Z 445.971,A -85,B 0,C 180,E1 -6328.814,E2 -6328.814} C_VEL
LIN {X 0,Y 495.75,Z 445.975,A -85,B 0,C 180,E1 -6331.726,E2 -6331.726} C_VEL
LIN {X 0,Y 495.767,Z 445.958,A -85,B 0,C 180,E1 -6334.695,E2 -6334.695} C_VEL
LIN {X 0,Y 495.726,Z 445.985,A -85,B 0,C 180,E1 -6337.561,E2 -6337.561} C_VEL
LIN {X 0,Y 495.786,Z 445.975,A -85,B 0,C 180,E1 -6340.052,E2 -6340.052} C_VEL
LIN {X 0,Y 495.756,Z 445.983,A -85,B 0,C 180,E1 -6342.879,E2 -6342.879} C_VEL
LIN {X 0,Y 495.726,Z 445.983,A -85,B 0,C 180,E1 -6345.999,E2 -6345.999} C_VEL
LIN {X 0,Y 495.773,Z 445.983,A -85,B 0,C 180,E1 -6349.302,E2 -6349.302} C_VEL
LIN {X 0,Y 495.725,Z 445.983,A -85,B 0,C 180,E1 -6352.439,E2 -6352.439} C_VEL
LIN {X 0,Y 495.78,Z 445.981,A -85,B 0,C 180,E1 -6355.458,E2 -6355.458} C_VEL
LIN {X 0,Y 495.753,Z 445.979,A -85,B 0,C 180,E1 -6358.364,E2 -6358.364} C_VEL
LIN {X 0,Y 495.748,Z 445.98,A -85,B 0,C 180,E1 -6360.768,E2 -6360.768} C_VEL
LIN {X 0,Y 495.093,Z 446.067,A -85,B 0,C 180,E1 -6361.447,E2 -6361.447} C_VEL
LIN {X 0,Y 492.24,Z 446.42,A -85,B 0,C 180,E1 -6362.549,E2 -6362.549} C_VEL
LIN {X 0,Y 489.833,Z 446.721,A -85,B 0,C 180,E1 -6363.438,E2 -6363.438} C_VEL
LIN {X 0,Y 488.816,Z 446.845,A -85,B 0,C 180,E1 -6364.124,E2 -6364.124} C_VEL
LIN {X 0,Y 488.742,Z 446.852,A -85,B 0,C 180,E1 -6364.357,E2 -6364.357} C_VEL
LIN {X 0,Y 488.723,Z 446.858,A -85,B 0,C 180,E1 -6367.154,E2 -6367.154} C_VEL
LIN {X 0,Y 488.721,Z 446.86,A -85,B 0,C 180,E1 -6369.811,E2 -6369.811} C_VEL
LIN {X 0,Y 488.73,Z 446.854,A -85,B 0,C 180,E1 -6372.424,E2 -6372.424} C_VEL
LIN {X 0,Y 488.758,Z 446.852,A -85,B 0,C 180,E1 -6375,E2 -6375} C_VEL
LIN {X 0,Y 488.826,Z 446.845,A -85,B 0,C 180,E1 -6378.388,E2 -6378.388} C_VEL
LIN {X 0,Y 488.814,Z 446.849,A -85,B 0,C 180,E1 -6381.734,E2 -6381.734} C_VEL
LIN {X 0,Y 488.851,Z 446.844,A -85,B 0,C 180,E1 -6384.224,E2 -6384.224} C_VEL
LIN {X 0,Y 488.958,Z 446.83,A -85,B 0,C 180,E1 -6387.529,E2 -6387.529} C_VEL
LIN {X 0,Y 488.951,Z 446.828,A -85,B 0,C 180,E1 -6390.824,E2 -6390.824} C_VEL
LIN {X 0,Y 488.958,Z 446.83,A -85,B 0,C 180,E1 -6392.471,E2 -6392.471} C_VEL
LIN {X 0,Y 488.851,Z 446.844,A -85,B 0,C 180,E1 -6395.776,E2 -6395.776} C_VEL
LIN {X 0,Y 488.814,Z 446.849,A -85,B 0,C 180,E1 -6398.266,E2 -6398.266} C_VEL
LIN {X 0,Y 488.826,Z 446.845,A -85,B 0,C 180,E1 -6401.612,E2 -6401.612} C_VEL
LIN {X 0,Y 488.758,Z 446.852,A -85,B 0,C 180,E1 -6405,E2 -6405} C_VEL
LIN {X 0,Y 488.751,Z 446.856,A -85,B 0,C 180,E1 -6408.442,E2 -6408.442} C_VEL
LIN {X 0,Y 488.702,Z 446.858,A -85,B 0,C 180,E1 -6411.07,E2 -6411.07} C_VEL
LIN {X 0,Y 488.684,Z 446.862,A -85,B 0,C 180,E1 -6413.745,E2 -6413.745} C_VEL
LIN {X 0,Y 488.794,Z 446.849,A -85,B 0,C 180,E1 -6416.945,E2 -6416.945} C_VEL
LIN {X 0,Y 488.704,Z 446.862,A -85,B 0,C 180,E1 -6420.363,E2 -6420.363} C_VEL
LIN {X 0,Y 488.73,Z 446.854,A -85,B 0,C 180,E1 -6423.484,E2 -6423.484} C_VEL
LIN {X 0,Y 488.682,Z 446.864,A -85,B 0,C 180,E1 -6426.355,E2 -6426.355} C_VEL
LIN {X 0,Y 488.735,Z 446.855,A -85,B 0,C 180,E1 -6429.25,E2 -6429.25} C_VEL
LIN {X 0,Y 488.704,Z 446.857,A -85,B 0,C 180,E1 -6431.6,E2 -6431.6} C_VEL
LIN {X 0,Y 488.704,Z 446.863,A -85,B 0,C 180,E1 -6434.801,E2 -6434.801} C_VEL
LIN {X 0,Y 488.726,Z 446.855,A -85,B 0,C 180,E1 -6437.479,E2 -6437.479} C_VEL
LIN {X 0,Y 488.741,Z 446.859,A -85,B 0,C 180,E1 -6440.75,E2 -6440.75} C_VEL
LIN {X 0,Y 488.677,Z 446.857,A -85,B 0,C 180,E1 -6443.868,E2 -6443.868} C_VEL
LIN {X 0,Y 488.73,Z 446.837,A -85,B 0,C 180,E1 -6446.877,E2 -6446.877} C_VEL
LIN {X 0,Y 488.725,Z 446.854,A -85,B 0,C 180,E1 -6449.781,E2 -6449.781} C_VEL
LIN {X 0,Y 488.79,Z 446.825,A -85,B 0,C 180,E1 -6453.054,E2 -6453.054} C_VEL
LIN {X 0,Y 488.684,Z 446.856,A -85,B 0,C 180,E1 -6456.254,E2 -6456.254} C_VEL
LIN {X 0,Y 488.736,Z 446.852,A -85,B 0,C 180,E1 -6459.176,E2 -6459.176} C_VEL
LIN {X 0,Y 488.749,Z 446.853,A -85,B 0,C 180,E1 -6461.628,E2 -6461.628} C_VEL
LIN {X 0,Y 488.755,Z 446.846,A -85,B 0,C 180,E1 -6465,E2 -6465} C_VEL
LIN {X 0,Y 488.798,Z 446.838,A -85,B 0,C 180,E1 -6468.388,E2 -6468.388} C_VEL
LIN {X 0,Y 488.809,Z 446.843,A -85,B 0,C 180,E1 -6471.734,E2 -6471.734} C_VEL
LIN {X 0,Y 488.855,Z 446.832,A -85,B 0,C 180,E1 -6474.224,E2 -6474.224} C_VEL
LIN {X 0,Y 488.952,Z 446.825,A -85,B 0,C 180,E1 -6477.529,E2 -6477.529} C_VEL
LIN {X 0,Y 488.946,Z 446.826,A -85,B 0,C 180,E1 -6480.824,E2 -6480.824} C_VEL
LIN {X 0,Y 488.953,Z 446.822,A -85,B 0,C 180,E1 -6482.472,E2 -6482.472} C_VEL
LIN {X 0,Y 488.846,Z 446.844,A -85,B 0,C 180,E1 -6485.776,E2 -6485.776} C_VEL
LIN {X 0,Y 488.809,Z 446.835,A -85,B 0,C 180,E1 -6488.267,E2 -6488.267} C_VEL
LIN {X 0,Y 488.799,Z 446.85,A -85,B 0,C 180,E1 -6491.613,E2 -6491.613} C_VEL
LIN {X 0,Y 488.753,Z 446.848,A -85,B 0,C 180,E1 -6495.001,E2 -6495.001} C_VEL
LIN {X 0,Y 488.746,Z 446.835,A -85,B 0,C 180,E1 -6498.443,E2 -6498.443} C_VEL
LIN {X 0,Y 488.698,Z 446.836,A -85,B 0,C 180,E1 -6501.071,E2 -6501.071} C_VEL
LIN {X 0,Y 488.685,Z 446.861,A -85,B 0,C 180,E1 -6503.746,E2 -6503.746} C_VEL
LIN {X 0,Y 488.791,Z 446.834,A -85,B 0,C 180,E1 -6506.946,E2 -6506.946} C_VEL
LIN {X 0,Y 488.711,Z 446.855,A -85,B 0,C 180,E1 -6510.365,E2 -6510.365} C_VEL
LIN {X 0,Y 488.728,Z 446.853,A -85,B 0,C 180,E1 -6513.485,E2 -6513.485} C_VEL
LIN {X 0,Y 488.682,Z 446.859,A -85,B 0,C 180,E1 -6516.356,E2 -6516.356} C_VEL
LIN {X 0,Y 488.736,Z 446.847,A -85,B 0,C 180,E1 -6519.251,E2 -6519.251} C_VEL
LIN {X 0,Y 488.725,Z 446.857,A -85,B 0,C 180,E1 -6522.522,E2 -6522.522} C_VEL
LIN {X 0,Y 488.706,Z 446.856,A -85,B 0,C 180,E1 -6525.199,E2 -6525.199} C_VEL
LIN {X 0,Y 488.703,Z 446.857,A -85,B 0,C 180,E1 -6528.401,E2 -6528.401} C_VEL
LIN {X 0,Y 488.699,Z 446.839,A -85,B 0,C 180,E1 -6530.948,E2 -6530.948} C_VEL
LIN {X 0,Y 488.681,Z 446.86,A -85,B 0,C 180,E1 -6533.869,E2 -6533.869} C_VEL
LIN {X 0,Y 488.732,Z 447.017,A -85,B 0,C 180,E1 -6534.953,E2 -6534.953} C_VEL
LIN {X 0,Y 491.826,Z 458.729,A -85,B 0,C 180,E1 -6537.112,E2 -6537.112} C_VEL
LIN {X 0,Y 494.232,Z 468.417,A -85,B 0,C 180,E1 -6538.801,E2 -6538.801} C_VEL
LIN {X 0,Y 493.619,Z 483.101,A -85,B 0,C 180,E1 -6541.022,E2 -6541.022} C_VEL
LIN {X 0,Y 499.769,Z 507.788,A -85,B 0,C 180,E1 -6541.827,E2 -6541.827} C_VEL
LIN {X 0,Y 498.127,Z 651.822,A -85,B 0,C 180,E1 -6544.008,E2 -6544.008} C_VEL
LIN {X 0,Y 497.521,Z 695.014,A -85,B 0,C 180,E1 -6544.679,E2 -6544.679} C_VEL
LIN {X 0,Y 497.153,Z 707.729,A -85,B 0,C 180,E1 -6544.963,E2 -6544.963} C_VEL
LIN {X 0,Y 496.729,Z 720.04,A -85,B 0,C 180,E1 -6545.331,E2 -6545.331} C_VEL
LIN {X 0,Y 496.121,Z 732.62,A -85,B 0,C 180,E1 -6545.8,E2 -6545.8} C_VEL
LIN {X 0,Y 495.519,Z 745.228,A -85,B 0,C 180,E1 -6546.38,E2 -6546.38} C_VEL
LIN {X 0,Y 494.82,Z 756.846,A -85,B 0,C 180,E1 -6547.01,E2 -6547.01} C_VEL
LIN {X 0,Y 494.144,Z 768.116,A -85,B 0,C 180,E1 -6547.721,E2 -6547.721} C_VEL
LIN {X 0,Y 493.32,Z 780.029,A -85,B 0,C 180,E1 -6548.589,E2 -6548.589} C_VEL
LIN {X 0,Y 492.593,Z 791.337,A -85,B 0,C 180,E1 -6549.541,E2 -6549.541} C_VEL
LIN {X 0,Y 491.724,Z 802.529,A -85,B 0,C 180,E1 -6550.614,E2 -6550.614} C_VEL
LIN {X 0,Y 491.075,Z 812.009,A -85,B 0,C 180,E1 -6551.649,E2 -6551.649} C_VEL
LIN {X 0,Y 490.358,Z 822.148,A -85,B 0,C 180,E1 -6552.914,E2 -6552.914} C_VEL
LIN {X 0,Y 489.812,Z 831.035,A -85,B 0,C 180,E1 -6554.18,E2 -6554.18} C_VEL
LIN {X 0,Y 489.31,Z 838.861,A -85,B 0,C 180,E1 -6555.443,E2 -6555.443} C_VEL
LIN {X 0,Y 488.965,Z 845.758,A -85,B 0,C 180,E1 -6556.705,E2 -6556.705} C_VEL
LIN {X 0,Y 488.676,Z 851.759,A -85,B 0,C 180,E1 -6557.946,E2 -6557.946} C_VEL
LIN {X 0,Y 488.325,Z 858.702,A -85,B 0,C 180,E1 -6559.636,E2 -6559.636} C_VEL
LIN {X 0,Y 488.104,Z 864.381,A -85,B 0,C 180,E1 -6561.305,E2 -6561.305} C_VEL
LIN {X 0,Y 488.053,Z 867.944,A -85,B 0,C 180,E1 -6562.554,E2 -6562.554} C_VEL
LIN {X 0,Y 487.958,Z 871.737,A -85,B 0,C 180,E1 -6564.214,E2 -6564.214} C_VEL
LIN {X 0,Y 487.882,Z 874.532,A -85,B 0,C 180,E1 -6565.87,E2 -6565.87} C_VEL
LIN {X 0,Y 487.945,Z 875.646,A -85,B 0,C 180,E1 -6566.697,E2 -6566.697} C_VEL
LIN {X 0,Y 487.883,Z 877.033,A -85,B 0,C 180,E1 -6568.349,E2 -6568.349} C_VEL
LIN {X 0,Y 487.814,Z 877.5,A -85,B 0,C 180,E1 -6570,E2 -6570} C_VEL
LIN {X 0,Y 487.883,Z 877.033,A -85,B 0,C 180,E1 -6571.651,E2 -6571.651} C_VEL
LIN {X 0,Y 487.945,Z 875.646,A -85,B 0,C 180,E1 -6573.303,E2 -6573.303} C_VEL
LIN {X 0,Y 487.907,Z 873.312,A -85,B 0,C 180,E1 -6574.958,E2 -6574.958} C_VEL
LIN {X 0,Y 488.028,Z 869.991,A -85,B 0,C 180,E1 -6576.615,E2 -6576.615} C_VEL
LIN {X 0,Y 488.085,Z 865.65,A -85,B 0,C 180,E1 -6578.279,E2 -6578.279} C_VEL
LIN {X 0,Y 488.213,Z 860.227,A -85,B 0,C 180,E1 -6579.947,E2 -6579.947} C_VEL
LIN {X 0,Y 488.447,Z 855.425,A -85,B 0,C 180,E1 -6581.2,E2 -6581.2} C_VEL
LIN {X 0,Y 488.839,Z 847.843,A -85,B 0,C 180,E1 -6582.876,E2 -6582.876} C_VEL
LIN {X 0,Y 489.181,Z 841.257,A -85,B 0,C 180,E1 -6584.136,E2 -6584.136} C_VEL
LIN {X 0,Y 489.687,Z 833.77,A -85,B 0,C 180,E1 -6585.397,E2 -6585.397} C_VEL
LIN {X 0,Y 490.186,Z 825.257,A -85,B 0,C 180,E1 -6586.663,E2 -6586.663} C_VEL
LIN {X 0,Y 490.847,Z 815.537,A -85,B 0,C 180,E1 -6587.929,E2 -6587.929} C_VEL
LIN {X 0,Y 491.559,Z 805.344,A -85,B 0,C 180,E1 -6589.089,E2 -6589.089} C_VEL
LIN {X 0,Y 492.312,Z 794.77,A -85,B 0,C 180,E1 -6590.144,E2 -6590.144} C_VEL
LIN {X 0,Y 493.025,Z 783.948,A -85,B 0,C 180,E1 -6591.096,E2 -6591.096} C_VEL
LIN {X 0,Y 493.842,Z 772.824,A -85,B 0,C 180,E1 -6591.948,E2 -6591.948} C_VEL
LIN {X 0,Y 494.566,Z 762.077,A -85,B 0,C 180,E1 -6592.672,E2 -6592.672} C_VEL
LIN {X 0,Y 495.28,Z 749.334,A -85,B 0,C 180,E1 -6593.41,E2 -6593.41} C_VEL
LIN {X 0,Y 496.014,Z 736.329,A -85,B 0,C 180,E1 -6594.038,E2 -6594.038} C_VEL
LIN {X 0,Y 496.597,Z 723.107,A -85,B 0,C 180,E1 -6594.564,E2 -6594.564} C_VEL
LIN {X 0,Y 497.101,Z 709.729,A -85,B 0,C 180,E1 -6594.984,E2 -6594.984} C_VEL
LIN {X 0,Y 497.517,Z 696.016,A -85,B 0,C 180,E1 -6595.302,E2 -6595.302} C_VEL
LIN {X 0,Y 498.077,Z 655.404,A -85,B 0,C 180,E1 -6595.939,E2 -6595.939} C_VEL
LIN {X 0,Y 499.8,Z 507.653,A -85,B 0,C 180,E1 -6598.174,E2 -6598.174} C_VEL
LIN {X 0,Y 493.617,Z 483.065,A -85,B 0,C 180,E1 -6598.978,E2 -6598.978} C_VEL
LIN {X 0,Y 494.327,Z 469.727,A -85,B 0,C 180,E1 -6600.989,E2 -6600.989} C_VEL
LIN {X 0,Y 493.088,Z 463.642,A -85,B 0,C 180,E1 -6602.023,E2 -6602.023} C_VEL
LIN {X 0,Y 489.382,Z 449.521,A -85,B 0,C 180,E1 -6604.558,E2 -6604.558} C_VEL
LIN {X 0,Y 488.76,Z 447.08,A -85,B 0,C 180,E1 -6605.037,E2 -6605.037} C_VEL
LIN {X 0,Y 488.685,Z 446.852,A -85,B 0,C 180,E1 -6606.355,E2 -6606.355} C_VEL
LIN {X 0,Y 488.696,Z 446.844,A -85,B 0,C 180,E1 -6609.254,E2 -6609.254} C_VEL
LIN {X 0,Y 488.702,Z 446.857,A -85,B 0,C 180,E1 -6611.599,E2 -6611.599} C_VEL
LIN {X 0,Y 488.706,Z 446.856,A -85,B 0,C 180,E1 -6614.801,E2 -6614.801} C_VEL
LIN {X 0,Y 488.725,Z 446.857,A -85,B 0,C 180,E1 -6617.478,E2 -6617.478} C_VEL
LIN {X 0,Y 488.736,Z 446.847,A -85,B 0,C 180,E1 -6620.749,E2 -6620.749} C_VEL
LIN {X 0,Y 488.679,Z 446.855,A -85,B 0,C 180,E1 -6623.868,E2 -6623.868} C_VEL
LIN {X 0,Y 488.732,Z 446.851,A -85,B 0,C 180,E1 -6626.877,E2 -6626.877} C_VEL
LIN {X 0,Y 488.726,Z 446.849,A -85,B 0,C 180,E1 -6629.781,E2 -6629.781} C_VEL
LIN {X 0,Y 488.791,Z 446.833,A -85,B 0,C 180,E1 -6633.054,E2 -6633.054} C_VEL
LIN {X 0,Y 488.685,Z 446.861,A -85,B 0,C 180,E1 -6636.254,E2 -6636.254} C_VEL
LIN {X 0,Y 488.737,Z 446.83,A -85,B 0,C 180,E1 -6639.175,E2 -6639.175} C_VEL
LIN {X 0,Y 488.726,Z 446.851,A -85,B 0,C 180,E1 -6642.423,E2 -6642.423} C_VEL
LIN {X 0,Y 488.753,Z 446.848,A -85,B 0,C 180,E1 -6644.999,E2 -6644.999} C_VEL
LIN {X 0,Y 488.799,Z 446.85,A -85,B 0,C 180,E1 -6648.387,E2 -6648.387} C_VEL
LIN {X 0,Y 488.809,Z 446.835,A -85,B 0,C 180,E1 -6651.733,E2 -6651.733} C_VEL
LIN {X 0,Y 488.846,Z 446.844,A -85,B 0,C 180,E1 -6654.224,E2 -6654.224} C_VEL
LIN {X 0,Y 488.953,Z 446.821,A -85,B 0,C 180,E1 -6657.528,E2 -6657.528} C_VEL
LIN {X 0,Y 488.946,Z 446.82,A -85,B 0,C 180,E1 -6660.823,E2 -6660.823} C_VEL
LIN {X 0,Y 488.952,Z 446.823,A -85,B 0,C 180,E1 -6662.471,E2 -6662.471} C_VEL
LIN {X 0,Y 488.855,Z 446.831,A -85,B 0,C 180,E1 -6665.776,E2 -6665.776} C_VEL
LIN {X 0,Y 488.809,Z 446.843,A -85,B 0,C 180,E1 -6668.266,E2 -6668.266} C_VEL
LIN {X 0,Y 488.798,Z 446.838,A -85,B 0,C 180,E1 -6671.612,E2 -6671.612} C_VEL
LIN {X 0,Y 488.755,Z 446.847,A -85,B 0,C 180,E1 -6675,E2 -6675} C_VEL
LIN {X 0,Y 488.745,Z 446.855,A -85,B 0,C 180,E1 -6678.442,E2 -6678.442} C_VEL
LIN {X 0,Y 488.698,Z 446.859,A -85,B 0,C 180,E1 -6681.071,E2 -6681.071} C_VEL
LIN {X 0,Y 488.684,Z 446.856,A -85,B 0,C 180,E1 -6683.746,E2 -6683.746} C_VEL
LIN {X 0,Y 488.79,Z 446.825,A -85,B 0,C 180,E1 -6686.946,E2 -6686.946} C_VEL
LIN {X 0,Y 488.71,Z 446.857,A -85,B 0,C 180,E1 -6690.365,E2 -6690.365} C_VEL
LIN {X 0,Y 488.727,Z 446.833,A -85,B 0,C 180,E1 -6693.485,E2 -6693.485} C_VEL
LIN {X 0,Y 488.681,Z 446.857,A -85,B 0,C 180,E1 -6696.356,E2 -6696.356} C_VEL
LIN {X 0,Y 488.741,Z 446.859,A -85,B 0,C 180,E1 -6699.25,E2 -6699.25} C_VEL
LIN {X 0,Y 488.726,Z 446.855,A -85,B 0,C 180,E1 -6702.521,E2 -6702.521} C_VEL
LIN {X 0,Y 488.704,Z 446.863,A -85,B 0,C 180,E1 -6705.199,E2 -6705.199} C_VEL
LIN {X 0,Y 488.704,Z 446.857,A -85,B 0,C 180,E1 -6708.4,E2 -6708.4} C_VEL
LIN {X 0,Y 488.734,Z 446.857,A -85,B 0,C 180,E1 -6710.942,E2 -6710.942} C_VEL
LIN {X 0,Y 488.679,Z 446.862,A -85,B 0,C 180,E1 -6713.869,E2 -6713.869} C_VEL
LIN {X 0,Y 488.734,Z 446.856,A -85,B 0,C 180,E1 -6716.878,E2 -6716.878} C_VEL
LIN {X 0,Y 488.718,Z 446.859,A -85,B 0,C 180,E1 -6719.781,E2 -6719.781} C_VEL
LIN {X 0,Y 488.794,Z 446.849,A -85,B 0,C 180,E1 -6723.055,E2 -6723.055} C_VEL
LIN {X 0,Y 488.742,Z 446.852,A -85,B 0,C 180,E1 -6724.357,E2 -6724.357} C_VEL
LIN {X 0,Y 488.095,Z 446.936,A -85,B 0,C 180,E1 -6725.045,E2 -6725.045} C_VEL
LIN {X 0,Y 485.227,Z 447.297,A -85,B 0,C 180,E1 -6726.161,E2 -6726.161} C_VEL
LIN {X 0,Y 482.781,Z 447.603,A -85,B 0,C 180,E1 -6727.061,E2 -6727.061} C_VEL
LIN {X 0,Y 481.723,Z 447.733,A -85,B 0,C 180,E1 -6727.756,E2 -6727.756} C_VEL
LIN {X 0,Y 481.634,Z 447.74,A -85,B 0,C 180,E1 -6727.992,E2 -6727.992} C_VEL
LIN {X 0,Y 481.701,Z 447.732,A -85,B 0,C 180,E1 -6730.393,E2 -6730.393} C_VEL
LIN {X 0,Y 481.687,Z 447.732,A -85,B 0,C 180,E1 -6733.034,E2 -6733.034} C_VEL
LIN {X 0,Y 481.686,Z 447.736,A -85,B 0,C 180,E1 -6735.639,E2 -6735.639} C_VEL
LIN {X 0,Y 481.791,Z 447.721,A -85,B 0,C 180,E1 -6738.216,E2 -6738.216} C_VEL
LIN {X 0,Y 481.759,Z 447.726,A -85,B 0,C 180,E1 -6741.612,E2 -6741.612} C_VEL
LIN {X 0,Y 481.812,Z 447.721,A -85,B 0,C 180,E1 -6744.14,E2 -6744.14} C_VEL
LIN {X 0,Y 481.925,Z 447.706,A -85,B 0,C 180,E1 -6747.493,E2 -6747.493} C_VEL
LIN {X 0,Y 481.902,Z 447.706,A -85,B 0,C 180,E1 -6750.836,E2 -6750.836} C_VEL
LIN {X 0,Y 481.925,Z 447.706,A -85,B 0,C 180,E1 -6752.507,E2 -6752.507} C_VEL
LIN {X 0,Y 481.812,Z 447.721,A -85,B 0,C 180,E1 -6755.86,E2 -6755.86} C_VEL
LIN {X 0,Y 481.759,Z 447.726,A -85,B 0,C 180,E1 -6758.388,E2 -6758.388} C_VEL
LIN {X 0,Y 481.791,Z 447.722,A -85,B 0,C 180,E1 -6761.784,E2 -6761.784} C_VEL
LIN {X 0,Y 481.739,Z 447.726,A -85,B 0,C 180,E1 -6765.224,E2 -6765.224} C_VEL
LIN {X 0,Y 481.708,Z 447.733,A -85,B 0,C 180,E1 -6768.721,E2 -6768.721} C_VEL
LIN {X 0,Y 481.64,Z 447.737,A -85,B 0,C 180,E1 -6771.394,E2 -6771.394} C_VEL
LIN {X 0,Y 481.669,Z 447.738,A -85,B 0,C 180,E1 -6774.113,E2 -6774.113} C_VEL
LIN {X 0,Y 481.747,Z 447.726,A -85,B 0,C 180,E1 -6777.14,E2 -6777.14} C_VEL
LIN {X 0,Y 481.673,Z 447.734,A -85,B 0,C 180,E1 -6779.741,E2 -6779.741} C_VEL
LIN {X 0,Y 481.667,Z 447.738,A -85,B 0,C 180,E1 -6782.674,E2 -6782.674} C_VEL
LIN {X 0,Y 481.637,Z 447.737,A -85,B 0,C 180,E1 -6785.709,E2 -6785.709} C_VEL
LIN {X 0,Y 481.707,Z 447.73,A -85,B 0,C 180,E1 -6789.353,E2 -6789.353} C_VEL
LIN {X 0,Y 481.641,Z 447.739,A -85,B 0,C 180,E1 -6792.16,E2 -6792.16} C_VEL
LIN {X 0,Y 481.652,Z 447.736,A -85,B 0,C 180,E1 -6795.542,E2 -6795.542} C_VEL
LIN {X 0,Y 481.668,Z 447.734,A -85,B 0,C 180,E1 -6798.084,E2 -6798.084} C_VEL
LIN {X 0,Y 481.695,Z 447.735,A -85,B 0,C 180,E1 -6801.144,E2 -6801.144} C_VEL
LIN {X 0,Y 481.659,Z 447.721,A -85,B 0,C 180,E1 -6804.794,E2 -6804.794} C_VEL
LIN {X 0,Y 481.664,Z 447.726,A -85,B 0,C 180,E1 -6807.326,E2 -6807.326} C_VEL
LIN {X 0,Y 481.679,Z 447.732,A -85,B 0,C 180,E1 -6810.259,E2 -6810.259} C_VEL
LIN {X 0,Y 481.743,Z 447.701,A -85,B 0,C 180,E1 -6813.112,E2 -6813.112} C_VEL
LIN {X 0,Y 481.668,Z 447.73,A -85,B 0,C 180,E1 -6815.887,E2 -6815.887} C_VEL
LIN {X 0,Y 481.693,Z 447.73,A -85,B 0,C 180,E1 -6819.027,E2 -6819.027} C_VEL
LIN {X 0,Y 481.698,Z 447.728,A -85,B 0,C 180,E1 -6822.158,E2 -6822.158} C_VEL
LIN {X 0,Y 481.734,Z 447.718,A -85,B 0,C 180,E1 -6824.776,E2 -6824.776} C_VEL
LIN {X 0,Y 481.743,Z 447.716,A -85,B 0,C 180,E1 -6828.215,E2 -6828.215} C_VEL
LIN {X 0,Y 481.754,Z 447.724,A -85,B 0,C 180,E1 -6831.612,E2 -6831.612} C_VEL
LIN {X 0,Y 481.815,Z 447.71,A -85,B 0,C 180,E1 -6834.14,E2 -6834.14} C_VEL
LIN {X 0,Y 481.919,Z 447.701,A -85,B 0,C 180,E1 -6837.493,E2 -6837.493} C_VEL
LIN {X 0,Y 481.897,Z 447.704,A -85,B 0,C 180,E1 -6840.836,E2 -6840.836} C_VEL
LIN {X 0,Y 481.92,Z 447.698,A -85,B 0,C 180,E1 -6842.508,E2 -6842.508} C_VEL
LIN {X 0,Y 481.807,Z 447.719,A -85,B 0,C 180,E1 -6845.861,E2 -6845.861} C_VEL
LIN {X 0,Y 481.755,Z 447.713,A -85,B 0,C 180,E1 -6848.389,E2 -6848.389} C_VEL
LIN {X 0,Y 481.743,Z 447.725,A -85,B 0,C 180,E1 -6851.785,E2 -6851.785} C_VEL
LIN {X 0,Y 481.733,Z 447.724,A -85,B 0,C 180,E1 -6855.225,E2 -6855.225} C_VEL
LIN {X 0,Y 481.703,Z 447.71,A -85,B 0,C 180,E1 -6858.722,E2 -6858.722} C_VEL
LIN {X 0,Y 481.637,Z 447.716,A -85,B 0,C 180,E1 -6861.395,E2 -6861.395} C_VEL
LIN {X 0,Y 481.669,Z 447.738,A -85,B 0,C 180,E1 -6864.114,E2 -6864.114} C_VEL
LIN {X 0,Y 481.744,Z 447.711,A -85,B 0,C 180,E1 -6867.141,E2 -6867.141} C_VEL
LIN {X 0,Y 481.68,Z 447.717,A -85,B 0,C 180,E1 -6869.741,E2 -6869.741} C_VEL
LIN {X 0,Y 481.666,Z 447.732,A -85,B 0,C 180,E1 -6872.675,E2 -6872.675} C_VEL
LIN {X 0,Y 481.636,Z 447.725,A -85,B 0,C 180,E1 -6875.71,E2 -6875.71} C_VEL
LIN {X 0,Y 481.708,Z 447.723,A -85,B 0,C 180,E1 -6879.354,E2 -6879.354} C_VEL
LIN {X 0,Y 481.667,Z 447.739,A -85,B 0,C 180,E1 -6882.158,E2 -6882.158} C_VEL
LIN {X 0,Y 481.654,Z 447.73,A -85,B 0,C 180,E1 -6884.458,E2 -6884.458} C_VEL
LIN {X 0,Y 481.642,Z 447.731,A -85,B 0,C 180,E1 -6887.84,E2 -6887.84} C_VEL
LIN {X 0,Y 481.657,Z 447.72,A -85,B 0,C 180,E1 -6890.654,E2 -6890.654} C_VEL
LIN {X 0,Y 481.626,Z 447.722,A -85,B 0,C 180,E1 -6893.376,E2 -6893.376} C_VEL
LIN {X 0,Y 481.67,Z 447.793,A -85,B 0,C 180,E1 -6894.509,E2 -6894.509} C_VEL
LIN {X 0,Y 483.424,Z 454.269,A -85,B 0,C 180,E1 -6895.782,E2 -6895.782} C_VEL
LIN {X 0,Y 487.323,Z 469.67,A -85,B 0,C 180,E1 -6898.551,E2 -6898.551} C_VEL
LIN {X 0,Y 487.425,Z 473.77,A -85,B 0,C 180,E1 -6899.213,E2 -6899.213} C_VEL
LIN {X 0,Y 486.933,Z 482.919,A -85,B 0,C 180,E1 -6900.591,E2 -6900.591} C_VEL
LIN {X 0,Y 493.467,Z 509.121,A -85,B 0,C 180,E1 -6901.459,E2 -6901.459} C_VEL
LIN {X 0,Y 491.797,Z 649.822,A -85,B 0,C 180,E1 -6903.619,E2 -6903.619} C_VEL
LIN {X 0,Y 491.091,Z 695.414,A -85,B 0,C 180,E1 -6904.335,E2 -6904.335} C_VEL
LIN {X 0,Y 490.692,Z 708.552,A -85,B 0,C 180,E1 -6904.64,E2 -6904.64} C_VEL
LIN {X 0,Y 490.153,Z 721.564,A -85,B 0,C 180,E1 -6905.042,E2 -6905.042} C_VEL
LIN {X 0,Y 489.55,Z 733.644,A -85,B 0,C 180,E1 -6905.511,E2 -6905.511} C_VEL
LIN {X 0,Y 488.919,Z 746.043,A -85,B 0,C 180,E1 -6906.098,E2 -6906.098} C_VEL
LIN {X 0,Y 488.134,Z 758.378,A -85,B 0,C 180,E1 -6906.788,E2 -6906.788} C_VEL
LIN {X 0,Y 487.343,Z 770.294,A -85,B 0,C 180,E1 -6907.571,E2 -6907.571} C_VEL
LIN {X 0,Y 486.526,Z 781.123,A -85,B 0,C 180,E1 -6908.386,E2 -6908.386} C_VEL
LIN {X 0,Y 485.766,Z 792.269,A -85,B 0,C 180,E1 -6909.351,E2 -6909.351} C_VEL
LIN {X 0,Y 484.864,Z 803.123,A -85,B 0,C 180,E1 -6910.417,E2 -6910.417} C_VEL
LIN {X 0,Y 484.089,Z 813.583,A -85,B 0,C 180,E1 -6911.593,E2 -6911.593} C_VEL
LIN {X 0,Y 483.48,Z 822.021,A -85,B 0,C 180,E1 -6912.663,E2 -6912.663} C_VEL
LIN {X 0,Y 482.859,Z 830.983,A -85,B 0,C 180,E1 -6913.946,E2 -6913.946} C_VEL
LIN {X 0,Y 482.355,Z 838.855,A -85,B 0,C 180,E1 -6915.228,E2 -6915.228} C_VEL
LIN {X 0,Y 481.956,Z 845.753,A -85,B 0,C 180,E1 -6916.508,E2 -6916.508} C_VEL
LIN {X 0,Y 481.615,Z 852.216,A -85,B 0,C 180,E1 -6917.877,E2 -6917.877} C_VEL
LIN {X 0,Y 481.292,Z 858.697,A -85,B 0,C 180,E1 -6919.483,E2 -6919.483} C_VEL
LIN {X 0,Y 481.041,Z 864.378,A -85,B 0,C 180,E1 -6921.176,E2 -6921.176} C_VEL
LIN {X 0,Y 480.976,Z 867.94,A -85,B 0,C 180,E1 -6922.443,E2 -6922.443} C_VEL
LIN {X 0,Y 480.869,Z 871.732,A -85,B 0,C 180,E1 -6924.128,E2 -6924.128} C_VEL
LIN {X 0,Y 480.785,Z 874.529,A -85,B 0,C 180,E1 -6925.809,E2 -6925.809} C_VEL
LIN {X 0,Y 480.85,Z 875.644,A -85,B 0,C 180,E1 -6926.648,E2 -6926.648} C_VEL
LIN {X 0,Y 480.784,Z 877.035,A -85,B 0,C 180,E1 -6928.325,E2 -6928.325} C_VEL
LIN {X 0,Y 480.738,Z 877.5,A -85,B 0,C 180,E1 -6930,E2 -6930} C_VEL
LIN {X 0,Y 480.784,Z 877.035,A -85,B 0,C 180,E1 -6931.675,E2 -6931.675} C_VEL
LIN {X 0,Y 480.85,Z 875.644,A -85,B 0,C 180,E1 -6933.352,E2 -6933.352} C_VEL
LIN {X 0,Y 480.833,Z 873.307,A -85,B 0,C 180,E1 -6935.031,E2 -6935.031} C_VEL
LIN {X 0,Y 480.951,Z 869.987,A -85,B 0,C 180,E1 -6936.713,E2 -6936.713} C_VEL
LIN {X 0,Y 481.012,Z 865.646,A -85,B 0,C 180,E1 -6938.401,E2 -6938.401} C_VEL
LIN {X 0,Y 481.167,Z 860.222,A -85,B 0,C 180,E1 -6940.094,E2 -6940.094} C_VEL
LIN {X 0,Y 481.404,Z 855.421,A -85,B 0,C 180,E1 -6941.366,E2 -6941.366} C_VEL
LIN {X 0,Y 481.824,Z 847.838,A -85,B 0,C 180,E1 -6943.066,E2 -6943.066} C_VEL
LIN {X 0,Y 482.203,Z 841.252,A -85,B 0,C 180,E1 -6944.345,E2 -6944.345} C_VEL
LIN {X 0,Y 482.757,Z 833.744,A -85,B 0,C 180,E1 -6945.624,E2 -6945.624} C_VEL
LIN {X 0,Y 483.285,Z 825.155,A -85,B 0,C 180,E1 -6946.908,E2 -6946.908} C_VEL
LIN {X 0,Y 483.976,Z 815.36,A -85,B 0,C 180,E1 -6948.192,E2 -6948.192} C_VEL
LIN {X 0,Y 484.814,Z 804.124,A -85,B 0,C 180,E1 -6949.476,E2 -6949.476} C_VEL
LIN {X 0,Y 485.639,Z 793.412,A -85,B 0,C 180,E1 -6950.544,E2 -6950.544} C_VEL
LIN {X 0,Y 486.329,Z 783.736,A -85,B 0,C 180,E1 -6951.4,E2 -6951.4} C_VEL
LIN {X 0,Y 487.227,Z 771.948,A -85,B 0,C 180,E1 -6952.312,E2 -6952.312} C_VEL
LIN {X 0,Y 488.01,Z 760.121,A -85,B 0,C 180,E1 -6953.106,E2 -6953.106} C_VEL
LIN {X 0,Y 488.788,Z 748.096,A -85,B 0,C 180,E1 -6953.796,E2 -6953.796} C_VEL
LIN {X 0,Y 489.572,Z 734.883,A -85,B 0,C 180,E1 -6954.432,E2 -6954.432} C_VEL
LIN {X 0,Y 490.148,Z 722.251,A -85,B 0,C 180,E1 -6954.933,E2 -6954.933} C_VEL
LIN {X 0,Y 490.682,Z 709.163,A -85,B 0,C 180,E1 -6955.344,E2 -6955.344} C_VEL
LIN {X 0,Y 491.1,Z 695.647,A -85,B 0,C 180,E1 -6955.659,E2 -6955.659} C_VEL
LIN {X 0,Y 491.742,Z 653.404,A -85,B 0,C 180,E1 -6956.327,E2 -6956.327} C_VEL
LIN {X 0,Y 493.474,Z 508.846,A -85,B 0,C 180,E1 -6958.545,E2 -6958.545} C_VEL
LIN {X 0,Y 486.916,Z 482.876,A -85,B 0,C 180,E1 -6959.41,E2 -6959.41} C_VEL
LIN {X 0,Y 487.537,Z 470.757,A -85,B 0,C 180,E1 -6961.261,E2 -6961.261} C_VEL
LIN {X 0,Y 483.949,Z 456.223,A -85,B 0,C 180,E1 -6963.857,E2 -6963.857} C_VEL
LIN {X 0,Y 481.743,Z 448.049,A -85,B 0,C 180,E1 -6965.413,E2 -6965.413} C_VEL
LIN {X 0,Y 481.653,Z 447.741,A -85,B 0,C 180,E1 -6965.707,E2 -6965.707} C_VEL
LIN {X 0,Y 481.666,Z 447.71,A -85,B 0,C 180,E1 -6968.858,E2 -6968.858} C_VEL
LIN {X 0,Y 481.647,Z 447.732,A -85,B 0,C 180,E1 -6971.912,E2 -6971.912} C_VEL
LIN {X 0,Y 481.654,Z 447.736,A -85,B 0,C 180,E1 -6974.457,E2 -6974.457} C_VEL
LIN {X 0,Y 481.682,Z 447.729,A -85,B 0,C 180,E1 -6976.845,E2 -6976.845} C_VEL
LIN {X 0,Y 481.682,Z 447.724,A -85,B 0,C 180,E1 -6980.06,E2 -6980.06} C_VEL
LIN {X 0,Y 481.623,Z 447.74,A -85,B 0,C 180,E1 -6983.253,E2 -6983.253} C_VEL
LIN {X 0,Y 481.702,Z 447.727,A -85,B 0,C 180,E1 -6986.329,E2 -6986.329} C_VEL
LIN {X 0,Y 481.651,Z 447.735,A -85,B 0,C 180,E1 -6989.415,E2 -6989.415} C_VEL
LIN {X 0,Y 481.694,Z 447.709,A -85,B 0,C 180,E1 -6992.168,E2 -6992.168} C_VEL
LIN {X 0,Y 481.71,Z 447.727,A -85,B 0,C 180,E1 -6994.969,E2 -6994.969} C_VEL
LIN {X 0,Y 481.642,Z 447.732,A -85,B 0,C 180,E1 -6997.704,E2 -6997.704} C_VEL
LIN {X 0,Y 481.697,Z 447.704,A -85,B 0,C 180,E1 -7000.393,E2 -7000.393} C_VEL
LIN {X 0,Y 481.683,Z 447.728,A -85,B 0,C 180,E1 -7003.034,E2 -7003.034} C_VEL
LIN {X 0,Y 481.68,Z 447.73,A -85,B 0,C 180,E1 -7005.638,E2 -7005.638} C_VEL
LIN {X 0,Y 481.743,Z 447.725,A -85,B 0,C 180,E1 -7008.215,E2 -7008.215} C_VEL
LIN {X 0,Y 481.755,Z 447.713,A -85,B 0,C 180,E1 -7011.611,E2 -7011.611} C_VEL
LIN {X 0,Y 481.807,Z 447.72,A -85,B 0,C 180,E1 -7014.139,E2 -7014.139} C_VEL
LIN {X 0,Y 481.92,Z 447.697,A -85,B 0,C 180,E1 -7017.492,E2 -7017.492} C_VEL
LIN {X 0,Y 481.897,Z 447.697,A -85,B 0,C 180,E1 -7020.835,E2 -7020.835} C_VEL
LIN {X 0,Y 481.919,Z 447.7,A -85,B 0,C 180,E1 -7022.507,E2 -7022.507} C_VEL
LIN {X 0,Y 481.815,Z 447.708,A -85,B 0,C 180,E1 -7025.86,E2 -7025.86} C_VEL
LIN {X 0,Y 481.754,Z 447.723,A -85,B 0,C 180,E1 -7028.388,E2 -7028.388} C_VEL
LIN {X 0,Y 481.743,Z 447.716,A -85,B 0,C 180,E1 -7031.785,E2 -7031.785} C_VEL
LIN {X 0,Y 481.734,Z 447.718,A -85,B 0,C 180,E1 -7035.224,E2 -7035.224} C_VEL
LIN {X 0,Y 481.703,Z 447.735,A -85,B 0,C 180,E1 -7038.722,E2 -7038.722} C_VEL
LIN {X 0,Y 481.638,Z 447.738,A -85,B 0,C 180,E1 -7041.395,E2 -7041.395} C_VEL
LIN {X 0,Y 481.668,Z 447.73,A -85,B 0,C 180,E1 -7044.113,E2 -7044.113} C_VEL
LIN {X 0,Y 481.743,Z 447.702,A -85,B 0,C 180,E1 -7047.141,E2 -7047.141} C_VEL
LIN {X 0,Y 481.679,Z 447.732,A -85,B 0,C 180,E1 -7049.741,E2 -7049.741} C_VEL
LIN {X 0,Y 481.664,Z 447.726,A -85,B 0,C 180,E1 -7052.674,E2 -7052.674} C_VEL
LIN {X 0,Y 481.634,Z 447.735,A -85,B 0,C 180,E1 -7055.709,E2 -7055.709} C_VEL
LIN {X 0,Y 481.712,Z 447.733,A -85,B 0,C 180,E1 -7059.355,E2 -7059.355} C_VEL
LIN {X 0,Y 481.667,Z 447.734,A -85,B 0,C 180,E1 -7062.158,E2 -7062.158} C_VEL
LIN {X 0,Y 481.652,Z 447.736,A -85,B 0,C 180,E1 -7064.458,E2 -7064.458} C_VEL
LIN {X 0,Y 481.641,Z 447.739,A -85,B 0,C 180,E1 -7067.84,E2 -7067.84} C_VEL
LIN {X 0,Y 481.707,Z 447.73,A -85,B 0,C 180,E1 -7070.647,E2 -7070.647} C_VEL
LIN {X 0,Y 481.637,Z 447.737,A -85,B 0,C 180,E1 -7074.291,E2 -7074.291} C_VEL
LIN {X 0,Y 481.667,Z 447.738,A -85,B 0,C 180,E1 -7077.326,E2 -7077.326} C_VEL
LIN {X 0,Y 481.673,Z 447.734,A -85,B 0,C 180,E1 -7080.259,E2 -7080.259} C_VEL
LIN {X 0,Y 481.747,Z 447.727,A -85,B 0,C 180,E1 -7083.113,E2 -7083.113} C_VEL
LIN {X 0,Y 481.673,Z 447.737,A -85,B 0,C 180,E1 -7085.887,E2 -7085.887} C_VEL
LIN {X 0,Y 481.634,Z 447.74,A -85,B 0,C 180,E1 -7087.992,E2 -7087.992} C_VEL
LIN {X 0,Y 480.965,Z 447.821,A -85,B 0,C 180,E1 -7088.69,E2 -7088.69} C_VEL
LIN {X 0,Y 478.136,Z 448.178,A -85,B 0,C 180,E1 -7089.824,E2 -7089.824} C_VEL
LIN {X 0,Y 475.752,Z 448.474,A -85,B 0,C 180,E1 -7090.738,E2 -7090.738} C_VEL
LIN {X 0,Y 474.732,Z 448.602,A -85,B 0,C 180,E1 -7091.444,E2 -7091.444} C_VEL
LIN {X 0,Y 474.651,Z 448.612,A -85,B 0,C 180,E1 -7091.683,E2 -7091.683} C_VEL
LIN {X 0,Y 474.696,Z 448.604,A -85,B 0,C 180,E1 -7094.545,E2 -7094.545} C_VEL
LIN {X 0,Y 474.735,Z 448.601,A -85,B 0,C 180,E1 -7098.039,E2 -7098.039} C_VEL
LIN {X 0,Y 474.724,Z 448.602,A -85,B 0,C 180,E1 -7101.487,E2 -7101.487} C_VEL
LIN {X 0,Y 474.775,Z 448.597,A -85,B 0,C 180,E1 -7104.052,E2 -7104.052} C_VEL
LIN {X 0,Y 474.891,Z 448.582,A -85,B 0,C 180,E1 -7107.455,E2 -7107.455} C_VEL
LIN {X 0,Y 474.909,Z 448.582,A -85,B 0,C 180,E1 -7110,E2 -7110} C_VEL
LIN {X 0,Y 474.891,Z 448.582,A -85,B 0,C 180,E1 -7112.545,E2 -7112.545} C_VEL
LIN {X 0,Y 474.775,Z 448.597,A -85,B 0,C 180,E1 -7115.948,E2 -7115.948} C_VEL
LIN {X 0,Y 474.724,Z 448.602,A -85,B 0,C 180,E1 -7118.513,E2 -7118.513} C_VEL
LIN {X 0,Y 474.735,Z 448.601,A -85,B 0,C 180,E1 -7121.961,E2 -7121.961} C_VEL
LIN {X 0,Y 474.677,Z 448.608,A -85,B 0,C 180,E1 -7125.768,E2 -7125.768} C_VEL
LIN {X 0,Y 474.661,Z 448.609,A -85,B 0,C 180,E1 -7129.01,E2 -7129.01} C_VEL
LIN {X 0,Y 474.583,Z 448.617,A -85,B 0,C 180,E1 -7131.729,E2 -7131.729} C_VEL
LIN {X 0,Y 474.652,Z 448.613,A -85,B 0,C 180,E1 -7134.493,E2 -7134.493} C_VEL
LIN {X 0,Y 474.694,Z 448.604,A -85,B 0,C 180,E1 -7137.338,E2 -7137.338} C_VEL
LIN {X 0,Y 474.599,Z 448.618,A -85,B 0,C 180,E1 -7140.81,E2 -7140.81} C_VEL
LIN {X 0,Y 474.632,Z 448.613,A -85,B 0,C 180,E1 -7143.984,E2 -7143.984} C_VEL
LIN {X 0,Y 474.569,Z 448.622,A -85,B 0,C 180,E1 -7146.9,E2 -7146.9} C_VEL
LIN {X 0,Y 474.643,Z 448.609,A -85,B 0,C 180,E1 -7149.651,E2 -7149.651} C_VEL
LIN {X 0,Y 474.607,Z 448.618,A -85,B 0,C 180,E1 -7152.934,E2 -7152.934} C_VEL
LIN {X 0,Y 474.61,Z 448.613,A -85,B 0,C 180,E1 -7155.896,E2 -7155.896} C_VEL
LIN {X 0,Y 474.639,Z 448.614,A -85,B 0,C 180,E1 -7159.038,E2 -7159.038} C_VEL
LIN {X 0,Y 474.612,Z 448.613,A -85,B 0,C 180,E1 -7161.702,E2 -7161.702} C_VEL
LIN {X 0,Y 474.621,Z 448.598,A -85,B 0,C 180,E1 -7164.726,E2 -7164.726} C_VEL
LIN {X 0,Y 474.628,Z 448.606,A -85,B 0,C 180,E1 -7167.788,E2 -7167.788} C_VEL
LIN {X 0,Y 474.623,Z 448.609,A -85,B 0,C 180,E1 -7170.883,E2 -7170.883} C_VEL
LIN {X 0,Y 474.657,Z 448.582,A -85,B 0,C 180,E1 -7173.629,E2 -7173.629} C_VEL
LIN {X 0,Y 474.626,Z 448.609,A -85,B 0,C 180,E1 -7176.641,E2 -7176.641} C_VEL
LIN {X 0,Y 474.647,Z 448.602,A -85,B 0,C 180,E1 -7180.09,E2 -7180.09} C_VEL
LIN {X 0,Y 474.641,Z 448.61,A -85,B 0,C 180,E1 -7182.774,E2 -7182.774} C_VEL
LIN {X 0,Y 474.642,Z 448.611,A -85,B 0,C 180,E1 -7185.421,E2 -7185.421} C_VEL
LIN {X 0,Y 474.696,Z 448.594,A -85,B 0,C 180,E1 -7188.038,E2 -7188.038} C_VEL
LIN {X 0,Y 474.719,Z 448.602,A -85,B 0,C 180,E1 -7191.487,E2 -7191.487} C_VEL
LIN {X 0,Y 474.776,Z 448.587,A -85,B 0,C 180,E1 -7194.053,E2 -7194.053} C_VEL
LIN {X 0,Y 474.886,Z 448.577,A -85,B 0,C 180,E1 -7197.456,E2 -7197.456} C_VEL
LIN {X 0,Y 474.848,Z 448.583,A -85,B 0,C 180,E1 -7200.848,E2 -7200.848} C_VEL
LIN {X 0,Y 474.886,Z 448.574,A -85,B 0,C 180,E1 -7202.545,E2 -7202.545} C_VEL
LIN {X 0,Y 474.77,Z 448.595,A -85,B 0,C 180,E1 -7205.948,E2 -7205.948} C_VEL
LIN {X 0,Y 474.72,Z 448.588,A -85,B 0,C 180,E1 -7208.514,E2 -7208.514} C_VEL
LIN {X 0,Y 474.696,Z 448.6,A -85,B 0,C 180,E1 -7211.963,E2 -7211.963} C_VEL
LIN {X 0,Y 474.691,Z 448.604,A -85,B 0,C 180,E1 -7215.456,E2 -7215.456} C_VEL
LIN {X 0,Y 474.656,Z 448.588,A -85,B 0,C 180,E1 -7219.011,E2 -7219.011} C_VEL
LIN {X 0,Y 474.58,Z 448.598,A -85,B 0,C 180,E1 -7221.729,E2 -7221.729} C_VEL
LIN {X 0,Y 474.651,Z 448.608,A -85,B 0,C 180,E1 -7224.493,E2 -7224.493} C_VEL
LIN {X 0,Y 474.691,Z 448.587,A -85,B 0,C 180,E1 -7227.339,E2 -7227.339} C_VEL
LIN {X 0,Y 474.603,Z 448.612,A -85,B 0,C 180,E1 -7230.812,E2 -7230.812} C_VEL
LIN {X 0,Y 474.631,Z 448.601,A -85,B 0,C 180,E1 -7233.984,E2 -7233.984} C_VEL
LIN {X 0,Y 474.569,Z 448.618,A -85,B 0,C 180,E1 -7236.901,E2 -7236.901} C_VEL
LIN {X 0,Y 474.644,Z 448.601,A -85,B 0,C 180,E1 -7239.652,E2 -7239.652} C_VEL
LIN {X 0,Y 474.645,Z 448.607,A -85,B 0,C 180,E1 -7242.931,E2 -7242.931} C_VEL
LIN {X 0,Y 474.603,Z 448.616,A -85,B 0,C 180,E1 -7245.896,E2 -7245.896} C_VEL
LIN {X 0,Y 474.623,Z 448.616,A -85,B 0,C 180,E1 -7249.041,E2 -7249.041} C_VEL
LIN {X 0,Y 474.605,Z 448.58,A -85,B 0,C 180,E1 -7251.705,E2 -7251.705} C_VEL
LIN {X 0,Y 474.62,Z 448.783,A -85,B 0,C 180,E1 -7254.141,E2 -7254.141} C_VEL
LIN {X 0,Y 477.957,Z 461.228,A -85,B 0,C 180,E1 -7256.525,E2 -7256.525} C_VEL
LIN {X 0,Y 480.64,Z 471.99,A -85,B 0,C 180,E1 -7258.484,E2 -7258.484} C_VEL
LIN {X 0,Y 480.579,Z 476.514,A -85,B 0,C 180,E1 -7259.214,E2 -7259.214} C_VEL
LIN {X 0,Y 480.246,Z 482.505,A -85,B 0,C 180,E1 -7260.13,E2 -7260.13} C_VEL
LIN {X 0,Y 487.252,Z 510.511,A -85,B 0,C 180,E1 -7261.087,E2 -7261.087} C_VEL
LIN {X 0,Y 485.359,Z 653.193,A -85,B 0,C 180,E1 -7263.3,E2 -7263.3} C_VEL
LIN {X 0,Y 484.687,Z 695.198,A -85,B 0,C 180,E1 -7263.971,E2 -7263.971} C_VEL
LIN {X 0,Y 484.237,Z 708.718,A -85,B 0,C 180,E1 -7264.288,E2 -7264.288} C_VEL
LIN {X 0,Y 483.661,Z 722.397,A -85,B 0,C 180,E1 -7264.722,E2 -7264.722} C_VEL
LIN {X 0,Y 482.979,Z 735.906,A -85,B 0,C 180,E1 -7265.27,E2 -7265.27} C_VEL
LIN {X 0,Y 482.068,Z 750.965,A -85,B 0,C 180,E1 -7266.023,E2 -7266.023} C_VEL
LIN {X 0,Y 480.967,Z 766.802,A -85,B 0,C 180,E1 -7267.009,E2 -7267.009} C_VEL
LIN {X 0,Y 480.001,Z 779.606,A -85,B 0,C 180,E1 -7267.964,E2 -7267.964} C_VEL
LIN {X 0,Y 479.102,Z 790.911,A -85,B 0,C 180,E1 -7268.938,E2 -7268.938} C_VEL
LIN {X 0,Y 478.161,Z 802.279,A -85,B 0,C 180,E1 -7270.061,E2 -7270.061} C_VEL
LIN {X 0,Y 477.404,Z 811.593,A -85,B 0,C 180,E1 -7271.103,E2 -7271.103} C_VEL
LIN {X 0,Y 476.604,Z 821.808,A -85,B 0,C 180,E1 -7272.405,E2 -7272.405} C_VEL
LIN {X 0,Y 475.934,Z 830.77,A -85,B 0,C 180,E1 -7273.706,E2 -7273.706} C_VEL
LIN {X 0,Y 475.386,Z 838.663,A -85,B 0,C 180,E1 -7275.006,E2 -7275.006} C_VEL
LIN {X 0,Y 474.948,Z 845.626,A -85,B 0,C 180,E1 -7276.305,E2 -7276.305} C_VEL
LIN {X 0,Y 474.577,Z 852.567,A -85,B 0,C 180,E1 -7277.792,E2 -7277.792} C_VEL
LIN {X 0,Y 474.232,Z 858.692,A -85,B 0,C 180,E1 -7279.325,E2 -7279.325} C_VEL
LIN {X 0,Y 473.987,Z 864.374,A -85,B 0,C 180,E1 -7281.044,E2 -7281.044} C_VEL
LIN {X 0,Y 473.896,Z 867.936,A -85,B 0,C 180,E1 -7282.33,E2 -7282.33} C_VEL
LIN {X 0,Y 473.785,Z 871.727,A -85,B 0,C 180,E1 -7284.04,E2 -7284.04} C_VEL
LIN {X 0,Y 473.693,Z 874.527,A -85,B 0,C 180,E1 -7285.746,E2 -7285.746} C_VEL
LIN {X 0,Y 473.743,Z 875.643,A -85,B 0,C 180,E1 -7286.598,E2 -7286.598} C_VEL
LIN {X 0,Y 473.689,Z 877.037,A -85,B 0,C 180,E1 -7288.3,E2 -7288.3} C_VEL
LIN {X 0,Y 473.664,Z 877.5,A -85,B 0,C 180,E1 -7290,E2 -7290} C_VEL
LIN {X 0,Y 473.689,Z 877.037,A -85,B 0,C 180,E1 -7291.7,E2 -7291.7} C_VEL
LIN {X 0,Y 473.743,Z 875.643,A -85,B 0,C 180,E1 -7293.402,E2 -7293.402} C_VEL
LIN {X 0,Y 473.761,Z 873.302,A -85,B 0,C 180,E1 -7295.106,E2 -7295.106} C_VEL
LIN {X 0,Y 473.882,Z 869.983,A -85,B 0,C 180,E1 -7296.814,E2 -7296.814} C_VEL
LIN {X 0,Y 473.955,Z 865.643,A -85,B 0,C 180,E1 -7298.527,E2 -7298.527} C_VEL
LIN {X 0,Y 474.132,Z 860.217,A -85,B 0,C 180,E1 -7300.246,E2 -7300.246} C_VEL
LIN {X 0,Y 474.373,Z 855.392,A -85,B 0,C 180,E1 -7301.537,E2 -7301.537} C_VEL
LIN {X 0,Y 474.82,Z 847.731,A -85,B 0,C 180,E1 -7303.263,E2 -7303.263} C_VEL
LIN {X 0,Y 475.207,Z 841.081,A -85,B 0,C 180,E1 -7304.561,E2 -7304.561} C_VEL
LIN {X 0,Y 475.818,Z 833.632,A -85,B 0,C 180,E1 -7305.841,E2 -7305.841} C_VEL
LIN {X 0,Y 476.372,Z 824.942,A -85,B 0,C 180,E1 -7307.161,E2 -7307.161} C_VEL
LIN {X 0,Y 477.128,Z 815.147,A -85,B 0,C 180,E1 -7308.462,E2 -7308.462} C_VEL
LIN {X 0,Y 477.909,Z 805.287,A -85,B 0,C 180,E1 -7309.616,E2 -7309.616} C_VEL
LIN {X 0,Y 478.798,Z 794.344,A -85,B 0,C 180,E1 -7310.739,E2 -7310.739} C_VEL
LIN {X 0,Y 479.641,Z 783.523,A -85,B 0,C 180,E1 -7311.714,E2 -7311.714} C_VEL
LIN {X 0,Y 480.556,Z 772.202,A -85,B 0,C 180,E1 -7312.603,E2 -7312.603} C_VEL
LIN {X 0,Y 481.415,Z 759.909,A -85,B 0,C 180,E1 -7313.441,E2 -7313.441} C_VEL
LIN {X 0,Y 482.231,Z 747.884,A -85,B 0,C 180,E1 -7314.14,E2 -7314.14} C_VEL
LIN {X 0,Y 483.067,Z 734.671,A -85,B 0,C 180,E1 -7314.782,E2 -7314.782} C_VEL
LIN {X 0,Y 483.7,Z 721.672,A -85,B 0,C 180,E1 -7315.303,E2 -7315.303} C_VEL
LIN {X 0,Y 484.294,Z 708.605,A -85,B 0,C 180,E1 -7315.712,E2 -7315.712} C_VEL
LIN {X 0,Y 484.697,Z 695.437,A -85,B 0,C 180,E1 -7316.024,E2 -7316.024} C_VEL
LIN {X 0,Y 485.34,Z 654.984,A -85,B 0,C 180,E1 -7316.672,E2 -7316.672} C_VEL
LIN {X 0,Y 487.289,Z 510.414,A -85,B 0,C 180,E1 -7318.912,E2 -7318.912} C_VEL
LIN {X 0,Y 480.229,Z 482.479,A -85,B 0,C 180,E1 -7319.872,E2 -7319.872} C_VEL
LIN {X 0,Y 480.781,Z 473.505,A -85,B 0,C 180,E1 -7321.26,E2 -7321.26} C_VEL
LIN {X 0,Y 479.538,Z 467.418,A -85,B 0,C 180,E1 -7322.338,E2 -7322.338} C_VEL
LIN {X 0,Y 475.889,Z 453.46,A -85,B 0,C 180,E1 -7324.929,E2 -7324.929} C_VEL
LIN {X 0,Y 474.632,Z 448.81,A -85,B 0,C 180,E1 -7325.862,E2 -7325.862} C_VEL
LIN {X 0,Y 474.607,Z 448.581,A -85,B 0,C 180,E1 -7328.457,E2 -7328.457} C_VEL
LIN {X 0,Y 474.615,Z 448.609,A -85,B 0,C 180,E1 -7331.785,E2 -7331.785} C_VEL
LIN {X 0,Y 474.615,Z 448.612,A -85,B 0,C 180,E1 -7334.702,E2 -7334.702} C_VEL
LIN {X 0,Y 474.642,Z 448.615,A -85,B 0,C 180,E1 -7337.759,E2 -7337.759} C_VEL
LIN {X 0,Y 474.662,Z 448.599,A -85,B 0,C 180,E1 -7340.456,E2 -7340.456} C_VEL
LIN {X 0,Y 474.587,Z 448.612,A -85,B 0,C 180,E1 -7343.676,E2 -7343.676} C_VEL
LIN {X 0,Y 474.636,Z 448.607,A -85,B 0,C 180,E1 -7346.779,E2 -7346.779} C_VEL
LIN {X 0,Y 474.606,Z 448.606,A -85,B 0,C 180,E1 -7349.77,E2 -7349.77} C_VEL
LIN {X 0,Y 474.707,Z 448.585,A -85,B 0,C 180,E1 -7352.68,E2 -7352.68} C_VEL
LIN {X 0,Y 474.651,Z 448.608,A -85,B 0,C 180,E1 -7355.507,E2 -7355.507} C_VEL
LIN {X 0,Y 474.661,Z 448.581,A -85,B 0,C 180,E1 -7359.185,E2 -7359.185} C_VEL
LIN {X 0,Y 474.648,Z 448.593,A -85,B 0,C 180,E1 -7361.884,E2 -7361.884} C_VEL
LIN {X 0,Y 474.691,Z 448.604,A -85,B 0,C 180,E1 -7364.544,E2 -7364.544} C_VEL
LIN {X 0,Y 474.696,Z 448.6,A -85,B 0,C 180,E1 -7368.037,E2 -7368.037} C_VEL
LIN {X 0,Y 474.72,Z 448.589,A -85,B 0,C 180,E1 -7371.486,E2 -7371.486} C_VEL
LIN {X 0,Y 474.77,Z 448.595,A -85,B 0,C 180,E1 -7374.052,E2 -7374.052} C_VEL
LIN {X 0,Y 474.886,Z 448.573,A -85,B 0,C 180,E1 -7377.455,E2 -7377.455} C_VEL
LIN {X 0,Y 474.902,Z 448.577,A -85,B 0,C 180,E1 -7380,E2 -7380} C_VEL
LIN {X 0,Y 474.886,Z 448.576,A -85,B 0,C 180,E1 -7382.544,E2 -7382.544} C_VEL
LIN {X 0,Y 474.776,Z 448.585,A -85,B 0,C 180,E1 -7385.947,E2 -7385.947} C_VEL
LIN {X 0,Y 474.719,Z 448.601,A -85,B 0,C 180,E1 -7388.513,E2 -7388.513} C_VEL
LIN {X 0,Y 474.696,Z 448.595,A -85,B 0,C 180,E1 -7391.962,E2 -7391.962} C_VEL
LIN {X 0,Y 474.691,Z 448.593,A -85,B 0,C 180,E1 -7395.456,E2 -7395.456} C_VEL
LIN {X 0,Y 474.656,Z 448.607,A -85,B 0,C 180,E1 -7399.01,E2 -7399.01} C_VEL
LIN {X 0,Y 474.58,Z 448.615,A -85,B 0,C 180,E1 -7401.729,E2 -7401.729} C_VEL
LIN {X 0,Y 474.65,Z 448.604,A -85,B 0,C 180,E1 -7404.493,E2 -7404.493} C_VEL
LIN {X 0,Y 474.69,Z 448.581,A -85,B 0,C 180,E1 -7407.339,E2 -7407.339} C_VEL
LIN {X 0,Y 474.601,Z 448.619,A -85,B 0,C 180,E1 -7410.812,E2 -7410.812} C_VEL
LIN {X 0,Y 474.629,Z 448.584,A -85,B 0,C 180,E1 -7413.984,E2 -7413.984} C_VEL
LIN {X 0,Y 474.569,Z 448.62,A -85,B 0,C 180,E1 -7416.9,E2 -7416.9} C_VEL
LIN {X 0,Y 474.647,Z 448.611,A -85,B 0,C 180,E1 -7419.652,E2 -7419.652} C_VEL
LIN {X 0,Y 474.644,Z 448.613,A -85,B 0,C 180,E1 -7422.93,E2 -7422.93} C_VEL
LIN {X 0,Y 474.602,Z 448.616,A -85,B 0,C 180,E1 -7425.895,E2 -7425.895} C_VEL
LIN {X 0,Y 474.634,Z 448.613,A -85,B 0,C 180,E1 -7429.039,E2 -7429.039} C_VEL
LIN {X 0,Y 474.61,Z 448.618,A -85,B 0,C 180,E1 -7431.703,E2 -7431.703} C_VEL
LIN {X 0,Y 474.624,Z 448.611,A -85,B 0,C 180,E1 -7434.727,E2 -7434.727} C_VEL
LIN {X 0,Y 474.632,Z 448.615,A -85,B 0,C 180,E1 -7437.788,E2 -7437.788} C_VEL
LIN {X 0,Y 474.619,Z 448.614,A -85,B 0,C 180,E1 -7440.885,E2 -7440.885} C_VEL
LIN {X 0,Y 474.662,Z 448.612,A -85,B 0,C 180,E1 -7443.629,E2 -7443.629} C_VEL
LIN {X 0,Y 474.631,Z 448.611,A -85,B 0,C 180,E1 -7446.641,E2 -7446.641} C_VEL
LIN {X 0,Y 474.65,Z 448.612,A -85,B 0,C 180,E1 -7450.09,E2 -7450.09} C_VEL
LIN {X 0,Y 474.651,Z 448.612,A -85,B 0,C 180,E1 -7451.683,E2 -7451.683} C_VEL
LIN {X 0,Y 473.989,Z 448.698,A -85,B 0,C 180,E1 -7452.392,E2 -7452.392} C_VEL
LIN {X 0,Y 471.138,Z 449.054,A -85,B 0,C 180,E1 -7453.543,E2 -7453.543} C_VEL
LIN {X 0,Y 468.721,Z 449.352,A -85,B 0,C 180,E1 -7454.472,E2 -7454.472} C_VEL
LIN {X 0,Y 467.68,Z 449.48,A -85,B 0,C 180,E1 -7455.189,E2 -7455.189} C_VEL
LIN {X 0,Y 467.593,Z 449.49,A -85,B 0,C 180,E1 -7455.432,E2 -7455.432} C_VEL
LIN {X 0,Y 467.667,Z 449.48,A -85,B 0,C 180,E1 -7458.734,E2 -7458.734} C_VEL
LIN {X 0,Y 467.745,Z 449.471,A -85,B 0,C 180,E1 -7462.228,E2 -7462.228} C_VEL
LIN {X 0,Y 467.721,Z 449.473,A -85,B 0,C 180,E1 -7464.828,E2 -7464.828} C_VEL
LIN {X 0,Y 467.857,Z 449.458,A -85,B 0,C 180,E1 -7467.417,E2 -7467.417} C_VEL
LIN {X 0,Y 467.88,Z 449.458,A -85,B 0,C 180,E1 -7470,E2 -7470} C_VEL
LIN {X 0,Y 467.857,Z 449.458,A -85,B 0,C 180,E1 -7472.583,E2 -7472.583} C_VEL
LIN {X 0,Y 467.74,Z 449.473,A -85,B 0,C 180,E1 -7476.037,E2 -7476.037} C_VEL
LIN {X 0,Y 467.678,Z 449.479,A -85,B 0,C 180,E1 -7478.643,E2 -7478.643} C_VEL
LIN {X 0,Y 467.679,Z 449.481,A -85,B 0,C 180,E1 -7482.145,E2 -7482.145} C_VEL
LIN {X 0,Y 467.646,Z 449.484,A -85,B 0,C 180,E1 -7485.885,E2 -7485.885} C_VEL
LIN {X 0,Y 467.619,Z 449.486,A -85,B 0,C 180,E1 -7489.307,E2 -7489.307} C_VEL
LIN {X 0,Y 467.53,Z 449.499,A -85,B 0,C 180,E1 -7492.074,E2 -7492.074} C_VEL
LIN {X 0,Y 467.597,Z 449.49,A -85,B 0,C 180,E1 -7494.887,E2 -7494.887} C_VEL
LIN {X 0,Y 467.622,Z 449.485,A -85,B 0,C 180,E1 -7497.768,E2 -7497.768} C_VEL
LIN {X 0,Y 467.563,Z 449.493,A -85,B 0,C 180,E1 -7501.045,E2 -7501.045} C_VEL
LIN {X 0,Y 467.584,Z 449.492,A -85,B 0,C 180,E1 -7504.242,E2 -7504.242} C_VEL
LIN {X 0,Y 467.544,Z 449.496,A -85,B 0,C 180,E1 -7507.186,E2 -7507.186} C_VEL
LIN {X 0,Y 467.588,Z 449.49,A -85,B 0,C 180,E1 -7510.262,E2 -7510.262} C_VEL
LIN {X 0,Y 467.579,Z 449.494,A -85,B 0,C 180,E1 -7512.567,E2 -7512.567} C_VEL
LIN {X 0,Y 467.563,Z 449.495,A -85,B 0,C 180,E1 -7515.053,E2 -7515.053} C_VEL
LIN {X 0,Y 467.617,Z 449.485,A -85,B 0,C 180,E1 -7517.444,E2 -7517.444} C_VEL
LIN {X 0,Y 467.611,Z 449.491,A -85,B 0,C 180,E1 -7520.859,E2 -7520.859} C_VEL
LIN {X 0,Y 467.554,Z 449.489,A -85,B 0,C 180,E1 -7524.26,E2 -7524.26} C_VEL
LIN {X 0,Y 467.573,Z 449.478,A -85,B 0,C 180,E1 -7527.321,E2 -7527.321} C_VEL
LIN {X 0,Y 467.57,Z 449.492,A -85,B 0,C 180,E1 -7530.665,E2 -7530.665} C_VEL
LIN {X 0,Y 467.618,Z 449.457,A -85,B 0,C 180,E1 -7533.2,E2 -7533.2} C_VEL
LIN {X 0,Y 467.583,Z 449.485,A -85,B 0,C 180,E1 -7536.468,E2 -7536.468} C_VEL
LIN {X 0,Y 467.614,Z 449.48,A -85,B 0,C 180,E1 -7539.777,E2 -7539.777} C_VEL
LIN {X 0,Y 467.6,Z 449.486,A -85,B 0,C 180,E1 -7542.507,E2 -7542.507} C_VEL
LIN {X 0,Y 467.599,Z 449.484,A -85,B 0,C 180,E1 -7545.197,E2 -7545.197} C_VEL
LIN {X 0,Y 467.647,Z 449.473,A -85,B 0,C 180,E1 -7547.855,E2 -7547.855} C_VEL
LIN {X 0,Y 467.673,Z 449.481,A -85,B 0,C 180,E1 -7551.357,E2 -7551.357} C_VEL
LIN {X 0,Y 467.739,Z 449.464,A -85,B 0,C 180,E1 -7553.963,E2 -7553.963} C_VEL
LIN {X 0,Y 467.851,Z 449.454,A -85,B 0,C 180,E1 -7557.417,E2 -7557.417} C_VEL
LIN {X 0,Y 467.872,Z 449.453,A -85,B 0,C 180,E1 -7560,E2 -7560} C_VEL
LIN {X 0,Y 467.851,Z 449.45,A -85,B 0,C 180,E1 -7562.583,E2 -7562.583} C_VEL
LIN {X 0,Y 467.734,Z 449.47,A -85,B 0,C 180,E1 -7566.038,E2 -7566.038} C_VEL
LIN {X 0,Y 467.673,Z 449.465,A -85,B 0,C 180,E1 -7568.643,E2 -7568.643} C_VEL
LIN {X 0,Y 467.648,Z 449.475,A -85,B 0,C 180,E1 -7572.146,E2 -7572.146} C_VEL
LIN {X 0,Y 467.63,Z 449.487,A -85,B 0,C 180,E1 -7575.695,E2 -7575.695} C_VEL
LIN {X 0,Y 467.608,Z 449.465,A -85,B 0,C 180,E1 -7578.765,E2 -7578.765} C_VEL
LIN {X 0,Y 467.571,Z 449.465,A -85,B 0,C 180,E1 -7581.268,E2 -7581.268} C_VEL
LIN {X 0,Y 467.566,Z 449.495,A -85,B 0,C 180,E1 -7583.944,E2 -7583.944} C_VEL
LIN {X 0,Y 467.619,Z 449.47,A -85,B 0,C 180,E1 -7586.8,E2 -7586.8} C_VEL
LIN {X 0,Y 467.579,Z 449.472,A -85,B 0,C 180,E1 -7589.736,E2 -7589.736} C_VEL
LIN {X 0,Y 467.577,Z 449.487,A -85,B 0,C 180,E1 -7592.759,E2 -7592.759} C_VEL
LIN {X 0,Y 467.55,Z 449.48,A -85,B 0,C 180,E1 -7595.89,E2 -7595.89} C_VEL
LIN {X 0,Y 467.609,Z 449.479,A -85,B 0,C 180,E1 -7599.142,E2 -7599.142} C_VEL
LIN {X 0,Y 467.613,Z 449.486,A -85,B 0,C 180,E1 -7602.572,E2 -7602.572} C_VEL
LIN {X 0,Y 467.565,Z 449.489,A -85,B 0,C 180,E1 -7605.054,E2 -7605.054} C_VEL
LIN {X 0,Y 467.584,Z 449.482,A -85,B 0,C 180,E1 -7607.441,E2 -7607.441} C_VEL
LIN {X 0,Y 467.555,Z 449.468,A -85,B 0,C 180,E1 -7610.854,E2 -7610.854} C_VEL
LIN {X 0,Y 467.58,Z 449.663,A -85,B 0,C 180,E1 -7613.714,E2 -7613.714} C_VEL
LIN {X 0,Y 471.071,Z 462.534,A -85,B 0,C 180,E1 -7616.239,E2 -7616.239} C_VEL
LIN {X 0,Y 473.988,Z 474.859,A -85,B 0,C 180,E1 -7618.509,E2 -7618.509} C_VEL
LIN {X 0,Y 473.589,Z 482.397,A -85,B 0,C 180,E1 -7619.677,E2 -7619.677} C_VEL
LIN {X 0,Y 481.114,Z 512.561,A -85,B 0,C 180,E1 -7620.72,E2 -7620.72} C_VEL
LIN {X 0,Y 478.433,Z 692.178,A -85,B 0,C 180,E1 -7623.547,E2 -7623.547} C_VEL
LIN {X 0,Y 477.976,Z 705.099,A -85,B 0,C 180,E1 -7623.826,E2 -7623.826} C_VEL
LIN {X 0,Y 477.445,Z 718.367,A -85,B 0,C 180,E1 -7624.224,E2 -7624.224} C_VEL
LIN {X 0,Y 476.785,Z 730.754,A -85,B 0,C 180,E1 -7624.693,E2 -7624.693} C_VEL
LIN {X 0,Y 476.053,Z 743.569,A -85,B 0,C 180,E1 -7625.294,E2 -7625.294} C_VEL
LIN {X 0,Y 475.117,Z 756.211,A -85,B 0,C 180,E1 -7625.998,E2 -7625.998} C_VEL
LIN {X 0,Y 474.294,Z 767.504,A -85,B 0,C 180,E1 -7626.737,E2 -7626.737} C_VEL
LIN {X 0,Y 473.326,Z 779.393,A -85,B 0,C 180,E1 -7627.637,E2 -7627.637} C_VEL
LIN {X 0,Y 472.392,Z 790.698,A -85,B 0,C 180,E1 -7628.624,E2 -7628.624} C_VEL
LIN {X 0,Y 471.446,Z 801.684,A -85,B 0,C 180,E1 -7629.721,E2 -7629.721} C_VEL
LIN {X 0,Y 470.577,Z 811.38,A -85,B 0,C 180,E1 -7630.819,E2 -7630.819} C_VEL
LIN {X 0,Y 469.722,Z 821.594,A -85,B 0,C 180,E1 -7632.139,E2 -7632.139} C_VEL
LIN {X 0,Y 469.02,Z 830.557,A -85,B 0,C 180,E1 -7633.459,E2 -7633.459} C_VEL
LIN {X 0,Y 468.449,Z 838.451,A -85,B 0,C 180,E1 -7634.779,E2 -7634.779} C_VEL
LIN {X 0,Y 467.945,Z 845.413,A -85,B 0,C 180,E1 -7636.096,E2 -7636.096} C_VEL
LIN {X 0,Y 467.515,Z 852.825,A -85,B 0,C 180,E1 -7637.72,E2 -7637.72} C_VEL
LIN {X 0,Y 467.184,Z 858.49,A -85,B 0,C 180,E1 -7639.162,E2 -7639.162} C_VEL
LIN {X 0,Y 466.899,Z 864.236,A -85,B 0,C 180,E1 -7640.906,E2 -7640.906} C_VEL
LIN {X 0,Y 466.813,Z 867.841,A -85,B 0,C 180,E1 -7642.213,E2 -7642.213} C_VEL
LIN {X 0,Y 466.707,Z 871.678,A -85,B 0,C 180,E1 -7643.949,E2 -7643.949} C_VEL
LIN {X 0,Y 466.606,Z 874.514,A -85,B 0,C 180,E1 -7645.681,E2 -7645.681} C_VEL
LIN {X 0,Y 466.638,Z 875.64,A -85,B 0,C 180,E1 -7646.546,E2 -7646.546} C_VEL
LIN {X 0,Y 466.598,Z 877.037,A -85,B 0,C 180,E1 -7648.274,E2 -7648.274} C_VEL
LIN {X 0,Y 466.565,Z 877.5,A -85,B 0,C 180,E1 -7650,E2 -7650} C_VEL
LIN {X 0,Y 466.598,Z 877.037,A -85,B 0,C 180,E1 -7651.726,E2 -7651.726} C_VEL
LIN {X 0,Y 466.638,Z 875.64,A -85,B 0,C 180,E1 -7653.454,E2 -7653.454} C_VEL
LIN {X 0,Y 466.669,Z 873.273,A -85,B 0,C 180,E1 -7655.184,E2 -7655.184} C_VEL
LIN {X 0,Y 466.814,Z 869.915,A -85,B 0,C 180,E1 -7656.917,E2 -7656.917} C_VEL
LIN {X 0,Y 466.878,Z 865.52,A -85,B 0,C 180,E1 -7658.658,E2 -7658.658} C_VEL
LIN {X 0,Y 467.067,Z 860.031,A -85,B 0,C 180,E1 -7660.402,E2 -7660.402} C_VEL
LIN {X 0,Y 467.342,Z 855.18,A -85,B 0,C 180,E1 -7661.713,E2 -7661.713} C_VEL
LIN {X 0,Y 467.754,Z 848.571,A -85,B 0,C 180,E1 -7663.246,E2 -7663.246} C_VEL
LIN {X 0,Y 468.232,Z 840.868,A -85,B 0,C 180,E1 -7664.783,E2 -7664.783} C_VEL
LIN {X 0,Y 468.856,Z 833.753,A -85,B 0,C 180,E1 -7666.029,E2 -7666.029} C_VEL
LIN {X 0,Y 469.464,Z 824.728,A -85,B 0,C 180,E1 -7667.421,E2 -7667.421} C_VEL
LIN {X 0,Y 470.277,Z 814.933,A -85,B 0,C 180,E1 -7668.741,E2 -7668.741} C_VEL
LIN {X 0,Y 471.049,Z 805.904,A -85,B 0,C 180,E1 -7669.82,E2 -7669.82} C_VEL
LIN {X 0,Y 471.984,Z 795.276,A -85,B 0,C 180,E1 -7670.938,E2 -7670.938} C_VEL
LIN {X 0,Y 472.951,Z 783.31,A -85,B 0,C 180,E1 -7672.037,E2 -7672.037} C_VEL
LIN {X 0,Y 473.894,Z 772.457,A -85,B 0,C 180,E1 -7672.903,E2 -7672.903} C_VEL
LIN {X 0,Y 474.746,Z 761.44,A -85,B 0,C 180,E1 -7673.675,E2 -7673.675} C_VEL
LIN {X 0,Y 475.692,Z 747.672,A -85,B 0,C 180,E1 -7674.494,E2 -7674.494} C_VEL
LIN {X 0,Y 476.571,Z 734.459,A -85,B 0,C 180,E1 -7675.144,E2 -7675.144} C_VEL
LIN {X 0,Y 477.234,Z 721.815,A -85,B 0,C 180,E1 -7675.657,E2 -7675.657} C_VEL
LIN {X 0,Y 477.885,Z 708.633,A -85,B 0,C 180,E1 -7676.076,E2 -7676.076} C_VEL
LIN {X 0,Y 478.327,Z 695.227,A -85,B 0,C 180,E1 -7676.397,E2 -7676.397} C_VEL
LIN {X 0,Y 479.059,Z 652.984,A -85,B 0,C 180,E1 -7677.08,E2 -7677.08} C_VEL
LIN {X 0,Y 481.043,Z 511.789,A -85,B 0,C 180,E1 -7679.297,E2 -7679.297} C_VEL
LIN {X 0,Y 473.617,Z 482.366,A -85,B 0,C 180,E1 -7680.322,E2 -7680.322} C_VEL
LIN {X 0,Y 473.985,Z 474.862,A -85,B 0,C 180,E1 -7681.491,E2 -7681.491} C_VEL
LIN {X 0,Y 471.427,Z 464.061,A -85,B 0,C 180,E1 -7683.476,E2 -7683.476} C_VEL
LIN {X 0,Y 468.136,Z 451.799,A -85,B 0,C 180,E1 -7685.837,E2 -7685.837} C_VEL
LIN {X 0,Y 467.553,Z 449.543,A -85,B 0,C 180,E1 -7686.355,E2 -7686.355} C_VEL
LIN {X 0,Y 467.555,Z 449.468,A -85,B 0,C 180,E1 -7689.146,E2 -7689.146} C_VEL
LIN {X 0,Y 467.581,Z 449.482,A -85,B 0,C 180,E1 -7692.566,E2 -7692.566} C_VEL
LIN {X 0,Y 467.565,Z 449.488,A -85,B 0,C 180,E1 -7695.053,E2 -7695.053} C_VEL
LIN {X 0,Y 467.604,Z 449.487,A -85,B 0,C 180,E1 -7697.442,E2 -7697.442} C_VEL
LIN {X 0,Y 467.609,Z 449.478,A -85,B 0,C 180,E1 -7700.858,E2 -7700.858} C_VEL
LIN {X 0,Y 467.556,Z 449.478,A -85,B 0,C 180,E1 -7704.26,E2 -7704.26} C_VEL
LIN {X 0,Y 467.575,Z 449.488,A -85,B 0,C 180,E1 -7707.32,E2 -7707.32} C_VEL
LIN {X 0,Y 467.569,Z 449.469,A -85,B 0,C 180,E1 -7710.665,E2 -7710.665} C_VEL
LIN {X 0,Y 467.619,Z 449.469,A -85,B 0,C 180,E1 -7713.2,E2 -7713.2} C_VEL
LIN {X 0,Y 467.585,Z 449.486,A -85,B 0,C 180,E1 -7716.468,E2 -7716.468} C_VEL
LIN {X 0,Y 467.614,Z 449.453,A -85,B 0,C 180,E1 -7719.777,E2 -7719.777} C_VEL
LIN {X 0,Y 467.6,Z 449.481,A -85,B 0,C 180,E1 -7722.506,E2 -7722.506} C_VEL
LIN {X 0,Y 467.597,Z 449.483,A -85,B 0,C 180,E1 -7725.196,E2 -7725.196} C_VEL
LIN {X 0,Y 467.648,Z 449.476,A -85,B 0,C 180,E1 -7727.854,E2 -7727.854} C_VEL
LIN {X 0,Y 467.673,Z 449.466,A -85,B 0,C 180,E1 -7731.357,E2 -7731.357} C_VEL
LIN {X 0,Y 467.734,Z 449.471,A -85,B 0,C 180,E1 -7733.962,E2 -7733.962} C_VEL
LIN {X 0,Y 467.851,Z 449.45,A -85,B 0,C 180,E1 -7737.417,E2 -7737.417} C_VEL
LIN {X 0,Y 467.872,Z 449.452,A -85,B 0,C 180,E1 -7740,E2 -7740} C_VEL
LIN {X 0,Y 467.851,Z 449.452,A -85,B 0,C 180,E1 -7742.583,E2 -7742.583} C_VEL
LIN {X 0,Y 467.739,Z 449.462,A -85,B 0,C 180,E1 -7746.037,E2 -7746.037} C_VEL
LIN {X 0,Y 467.673,Z 449.481,A -85,B 0,C 180,E1 -7748.643,E2 -7748.643} C_VEL
LIN {X 0,Y 467.647,Z 449.474,A -85,B 0,C 180,E1 -7752.145,E2 -7752.145} C_VEL
LIN {X 0,Y 467.629,Z 449.472,A -85,B 0,C 180,E1 -7755.695,E2 -7755.695} C_VEL
LIN {X 0,Y 467.608,Z 449.489,A -85,B 0,C 180,E1 -7758.765,E2 -7758.765} C_VEL
LIN {X 0,Y 467.571,Z 449.491,A -85,B 0,C 180,E1 -7761.268,E2 -7761.268} C_VEL
LIN {X 0,Y 467.564,Z 449.487,A -85,B 0,C 180,E1 -7763.943,E2 -7763.943} C_VEL
LIN {X 0,Y 467.618,Z 449.457,A -85,B 0,C 180,E1 -7766.8,E2 -7766.8} C_VEL
LIN {X 0,Y 467.578,Z 449.489,A -85,B 0,C 180,E1 -7769.736,E2 -7769.736} C_VEL
LIN {X 0,Y 467.575,Z 449.476,A -85,B 0,C 180,E1 -7772.759,E2 -7772.759} C_VEL
LIN {X 0,Y 467.548,Z 449.489,A -85,B 0,C 180,E1 -7775.89,E2 -7775.89} C_VEL
LIN {X 0,Y 467.611,Z 449.491,A -85,B 0,C 180,E1 -7779.141,E2 -7779.141} C_VEL
LIN {X 0,Y 467.611,Z 449.486,A -85,B 0,C 180,E1 -7782.572,E2 -7782.572} C_VEL
LIN {X 0,Y 467.563,Z 449.496,A -85,B 0,C 180,E1 -7785.053,E2 -7785.053} C_VEL
LIN {X 0,Y 467.581,Z 449.494,A -85,B 0,C 180,E1 -7787.44,E2 -7787.44} C_VEL
LIN {X 0,Y 467.608,Z 449.488,A -85,B 0,C 180,E1 -7790.859,E2 -7790.859} C_VEL
LIN {X 0,Y 467.557,Z 449.491,A -85,B 0,C 180,E1 -7794.261,E2 -7794.261} C_VEL
LIN {X 0,Y 467.576,Z 449.493,A -85,B 0,C 180,E1 -7797.321,E2 -7797.321} C_VEL
LIN {X 0,Y 467.564,Z 449.492,A -85,B 0,C 180,E1 -7800.668,E2 -7800.668} C_VEL
LIN {X 0,Y 467.623,Z 449.486,A -85,B 0,C 180,E1 -7803.201,E2 -7803.201} C_VEL
LIN {X 0,Y 467.588,Z 449.489,A -85,B 0,C 180,E1 -7806.468,E2 -7806.468} C_VEL
LIN {X 0,Y 467.618,Z 449.488,A -85,B 0,C 180,E1 -7809.777,E2 -7809.777} C_VEL
LIN {X 0,Y 467.605,Z 449.486,A -85,B 0,C 180,E1 -7812.507,E2 -7812.507} C_VEL
LIN {X 0,Y 467.593,Z 449.49,A -85,B 0,C 180,E1 -7815.432,E2 -7815.432} C_VEL
LIN {X 0,Y 466.926,Z 449.574,A -85,B 0,C 180,E1 -7816.151,E2 -7816.151} C_VEL
LIN {X 0,Y 464.091,Z 449.926,A -85,B 0,C 180,E1 -7817.32,E2 -7817.32} C_VEL
LIN {X 0,Y 461.696,Z 450.224,A -85,B 0,C 180,E1 -7818.262,E2 -7818.262} C_VEL
LIN {X 0,Y 460.667,Z 450.352,A -85,B 0,C 180,E1 -7818.99,E2 -7818.99} C_VEL
LIN {X 0,Y 460.583,Z 450.363,A -85,B 0,C 180,E1 -7819.236,E2 -7819.236} C_VEL
LIN {X 0,Y 460.716,Z 450.346,A -85,B 0,C 180,E1 -7822.539,E2 -7822.539} C_VEL
LIN {X 0,Y 460.694,Z 450.349,A -85,B 0,C 180,E1 -7824.748,E2 -7824.748} C_VEL
LIN {X 0,Y 460.822,Z 450.334,A -85,B 0,C 180,E1 -7827.378,E2 -7827.378} C_VEL
LIN {X 0,Y 460.85,Z 450.333,A -85,B 0,C 180,E1 -7830,E2 -7830} C_VEL
LIN {X 0,Y 460.822,Z 450.334,A -85,B 0,C 180,E1 -7832.622,E2 -7832.622} C_VEL
LIN {X 0,Y 460.706,Z 450.349,A -85,B 0,C 180,E1 -7836.13,E2 -7836.13} C_VEL
LIN {X 0,Y 460.625,Z 450.357,A -85,B 0,C 180,E1 -7838.776,E2 -7838.776} C_VEL
LIN {X 0,Y 460.63,Z 450.359,A -85,B 0,C 180,E1 -7842.457,E2 -7842.457} C_VEL
LIN {X 0,Y 460.596,Z 450.362,A -85,B 0,C 180,E1 -7845.997,E2 -7845.997} C_VEL
LIN {X 0,Y 460.566,Z 450.366,A -85,B 0,C 180,E1 -7848.902,E2 -7848.902} C_VEL
LIN {X 0,Y 460.511,Z 450.37,A -85,B 0,C 180,E1 -7851.485,E2 -7851.485} C_VEL
LIN {X 0,Y 460.537,Z 450.37,A -85,B 0,C 180,E1 -7854.332,E2 -7854.332} C_VEL
LIN {X 0,Y 460.579,Z 450.363,A -85,B 0,C 180,E1 -7857.243,E2 -7857.243} C_VEL
LIN {X 0,Y 460.505,Z 450.373,A -85,B 0,C 180,E1 -7860.24,E2 -7860.24} C_VEL
LIN {X 0,Y 460.523,Z 450.369,A -85,B 0,C 180,E1 -7863.324,E2 -7863.324} C_VEL
LIN {X 0,Y 460.473,Z 450.38,A -85,B 0,C 180,E1 -7866.529,E2 -7866.529} C_VEL
LIN {X 0,Y 460.568,Z 450.363,A -85,B 0,C 180,E1 -7869.857,E2 -7869.857} C_VEL
LIN {X 0,Y 460.506,Z 450.374,A -85,B 0,C 180,E1 -7872.9,E2 -7872.9} C_VEL
LIN {X 0,Y 460.516,Z 450.369,A -85,B 0,C 180,E1 -7875.828,E2 -7875.828} C_VEL
LIN {X 0,Y 460.536,Z 450.371,A -85,B 0,C 180,E1 -7878.99,E2 -7878.99} C_VEL
LIN {X 0,Y 460.539,Z 450.369,A -85,B 0,C 180,E1 -7881.269,E2 -7881.269} C_VEL
LIN {X 0,Y 460.505,Z 450.358,A -85,B 0,C 180,E1 -7884.554,E2 -7884.554} C_VEL
LIN {X 0,Y 460.524,Z 450.363,A -85,B 0,C 180,E1 -7887.715,E2 -7887.715} C_VEL
LIN {X 0,Y 460.539,Z 450.365,A -85,B 0,C 180,E1 -7890.769,E2 -7890.769} C_VEL
LIN {X 0,Y 460.559,Z 450.335,A -85,B 0,C 180,E1 -7893.735,E2 -7893.735} C_VEL
LIN {X 0,Y 460.537,Z 450.364,A -85,B 0,C 180,E1 -7896.624,E2 -7896.624} C_VEL
LIN {X 0,Y 460.542,Z 450.361,A -85,B 0,C 180,E1 -7899.453,E2 -7899.453} C_VEL
LIN {X 0,Y 460.55,Z 450.363,A -85,B 0,C 180,E1 -7902.23,E2 -7902.23} C_VEL
LIN {X 0,Y 460.557,Z 450.357,A -85,B 0,C 180,E1 -7904.965,E2 -7904.965} C_VEL
LIN {X 0,Y 460.604,Z 450.349,A -85,B 0,C 180,E1 -7908.559,E2 -7908.559} C_VEL
LIN {X 0,Y 460.686,Z 450.343,A -85,B 0,C 180,E1 -7912.109,E2 -7912.109} C_VEL
LIN {X 0,Y 460.694,Z 450.34,A -85,B 0,C 180,E1 -7914.749,E2 -7914.749} C_VEL
LIN {X 0,Y 460.816,Z 450.33,A -85,B 0,C 180,E1 -7917.378,E2 -7917.378} C_VEL
LIN {X 0,Y 460.843,Z 450.329,A -85,B 0,C 180,E1 -7920,E2 -7920} C_VEL
LIN {X 0,Y 460.816,Z 450.327,A -85,B 0,C 180,E1 -7922.623,E2 -7922.623} C_VEL
LIN {X 0,Y 460.7,Z 450.346,A -85,B 0,C 180,E1 -7926.13,E2 -7926.13} C_VEL
LIN {X 0,Y 460.621,Z 450.344,A -85,B 0,C 180,E1 -7928.776,E2 -7928.776} C_VEL
LIN {X 0,Y 460.604,Z 450.35,A -85,B 0,C 180,E1 -7932.445,E2 -7932.445} C_VEL
LIN {X 0,Y 460.591,Z 450.36,A -85,B 0,C 180,E1 -7935.998,E2 -7935.998} C_VEL
LIN {X 0,Y 460.562,Z 450.341,A -85,B 0,C 180,E1 -7938.902,E2 -7938.902} C_VEL
LIN {X 0,Y 460.507,Z 450.346,A -85,B 0,C 180,E1 -7941.486,E2 -7941.486} C_VEL
LIN {X 0,Y 460.535,Z 450.368,A -85,B 0,C 180,E1 -7944.333,E2 -7944.333} C_VEL
LIN {X 0,Y 460.576,Z 450.343,A -85,B 0,C 180,E1 -7947.244,E2 -7947.244} C_VEL
LIN {X 0,Y 460.519,Z 450.359,A -85,B 0,C 180,E1 -7950.239,E2 -7950.239} C_VEL
LIN {X 0,Y 460.522,Z 450.366,A -85,B 0,C 180,E1 -7953.325,E2 -7953.325} C_VEL
LIN {X 0,Y 460.473,Z 450.374,A -85,B 0,C 180,E1 -7956.53,E2 -7956.53} C_VEL
LIN {X 0,Y 460.57,Z 450.351,A -85,B 0,C 180,E1 -7959.858,E2 -7959.858} C_VEL
LIN {X 0,Y 460.537,Z 450.364,A -85,B 0,C 180,E1 -7962.905,E2 -7962.905} C_VEL
LIN {X 0,Y 460.506,Z 450.372,A -85,B 0,C 180,E1 -7965.831,E2 -7965.831} C_VEL
LIN {X 0,Y 460.525,Z 450.373,A -85,B 0,C 180,E1 -7968.989,E2 -7968.989} C_VEL
LIN {X 0,Y 460.514,Z 450.336,A -85,B 0,C 180,E1 -7971.267,E2 -7971.267} C_VEL
LIN {X 0,Y 460.543,Z 450.548,A -85,B 0,C 180,E1 -7973.273,E2 -7973.273} C_VEL
LIN {X 0,Y 464.125,Z 463.761,A -85,B 0,C 180,E1 -7975.926,E2 -7975.926} C_VEL
LIN {X 0,Y 467.124,Z 475.976,A -85,B 0,C 180,E1 -7978.226,E2 -7978.226} C_VEL
LIN {X 0,Y 467.013,Z 481.071,A -85,B 0,C 180,E1 -7979.068,E2 -7979.068} C_VEL
LIN {X 0,Y 467.009,Z 482.333,A -85,B 0,C 180,E1 -7979.215,E2 -7979.215} C_VEL
LIN {X 0,Y 474.822,Z 513.287,A -85,B 0,C 180,E1 -7980.31,E2 -7980.31} C_VEL
LIN {X 0,Y 472.51,Z 666.386,A -85,B 0,C 180,E1 -7982.741,E2 -7982.741} C_VEL
LIN {X 0,Y 471.932,Z 696.184,A -85,B 0,C 180,E1 -7983.242,E2 -7983.242} C_VEL
LIN {X 0,Y 471.304,Z 713.167,A -85,B 0,C 180,E1 -7983.674,E2 -7983.674} C_VEL
LIN {X 0,Y 470.394,Z 729.457,A -85,B 0,C 180,E1 -7984.273,E2 -7984.273} C_VEL
LIN {X 0,Y 469.541,Z 743.357,A -85,B 0,C 180,E1 -7984.927,E2 -7984.927} C_VEL
LIN {X 0,Y 468.579,Z 756,A -85,B 0,C 180,E1 -7985.641,E2 -7985.641} C_VEL
LIN {X 0,Y 467.607,Z 768.314,A -85,B 0,C 180,E1 -7986.464,E2 -7986.464} C_VEL
LIN {X 0,Y 466.558,Z 780.486,A -85,B 0,C 180,E1 -7987.412,E2 -7987.412} C_VEL
LIN {X 0,Y 465.67,Z 790.484,A -85,B 0,C 180,E1 -7988.3,E2 -7988.3} C_VEL
LIN {X 0,Y 464.663,Z 801.47,A -85,B 0,C 180,E1 -7989.412,E2 -7989.412} C_VEL
LIN {X 0,Y 463.769,Z 811.167,A -85,B 0,C 180,E1 -7990.526,E2 -7990.526} C_VEL
LIN {X 0,Y 462.831,Z 821.38,A -85,B 0,C 180,E1 -7991.864,E2 -7991.864} C_VEL
LIN {X 0,Y 462.092,Z 830.343,A -85,B 0,C 180,E1 -7993.204,E2 -7993.204} C_VEL
LIN {X 0,Y 461.503,Z 838.238,A -85,B 0,C 180,E1 -7994.544,E2 -7994.544} C_VEL
LIN {X 0,Y 460.929,Z 845.199,A -85,B 0,C 180,E1 -7995.88,E2 -7995.88} C_VEL
LIN {X 0,Y 460.54,Z 851.52,A -85,B 0,C 180,E1 -7997.261,E2 -7997.261} C_VEL
LIN {X 0,Y 460.137,Z 858.278,A -85,B 0,C 180,E1 -7998.994,E2 -7998.994} C_VEL
LIN {X 0,Y 459.824,Z 864.024,A -85,B 0,C 180,E1 -8000.765,E2 -8000.765} C_VEL
LIN {X 0,Y 459.727,Z 867.63,A -85,B 0,C 180,E1 -8002.092,E2 -8002.092} C_VEL
LIN {X 0,Y 459.636,Z 871.468,A -85,B 0,C 180,E1 -8003.856,E2 -8003.856} C_VEL
LIN {X 0,Y 459.521,Z 874.304,A -85,B 0,C 180,E1 -8005.614,E2 -8005.614} C_VEL
LIN {X 0,Y 459.557,Z 876.179,A -85,B 0,C 180,E1 -8007.37,E2 -8007.37} C_VEL
LIN {X 0,Y 459.51,Z 876.85,A -85,B 0,C 180,E1 -8008.247,E2 -8008.247} C_VEL
LIN {X 0,Y 459.469,Z 877.318,A -85,B 0,C 180,E1 -8010,E2 -8010} C_VEL
LIN {X 0,Y 459.51,Z 876.85,A -85,B 0,C 180,E1 -8011.753,E2 -8011.753} C_VEL
LIN {X 0,Y 459.534,Z 875.435,A -85,B 0,C 180,E1 -8013.507,E2 -8013.507} C_VEL
LIN {X 0,Y 459.582,Z 873.062,A -85,B 0,C 180,E1 -8015.264,E2 -8015.264} C_VEL
LIN {X 0,Y 459.723,Z 869.704,A -85,B 0,C 180,E1 -8017.025,E2 -8017.025} C_VEL
LIN {X 0,Y 459.811,Z 865.309,A -85,B 0,C 180,E1 -8018.792,E2 -8018.792} C_VEL
LIN {X 0,Y 460.016,Z 859.819,A -85,B 0,C 180,E1 -8020.564,E2 -8020.564} C_VEL
LIN {X 0,Y 460.307,Z 855.013,A -85,B 0,C 180,E1 -8021.883,E2 -8021.883} C_VEL
LIN {X 0,Y 460.8,Z 847.305,A -85,B 0,C 180,E1 -8023.674,E2 -8023.674} C_VEL
LIN {X 0,Y 461.263,Z 840.654,A -85,B 0,C 180,E1 -8025.012,E2 -8025.012} C_VEL
LIN {X 0,Y 461.949,Z 832.58,A -85,B 0,C 180,E1 -8026.433,E2 -8026.433} C_VEL
LIN {X 0,Y 462.588,Z 824.515,A -85,B 0,C 180,E1 -8027.689,E2 -8027.689} C_VEL
LIN {X 0,Y 463.44,Z 814.72,A -85,B 0,C 180,E1 -8029.028,E2 -8029.028} C_VEL
LIN {X 0,Y 464.302,Z 804.962,A -85,B 0,C 180,E1 -8030.204,E2 -8030.204} C_VEL
LIN {X 0,Y 465.357,Z 793.918,A -85,B 0,C 180,E1 -8031.367,E2 -8031.367} C_VEL
LIN {X 0,Y 466.282,Z 783.097,A -85,B 0,C 180,E1 -8032.369,E2 -8032.369} C_VEL
LIN {X 0,Y 467.357,Z 771.204,A -85,B 0,C 180,E1 -8033.323,E2 -8033.323} C_VEL
LIN {X 0,Y 468.292,Z 759.485,A -85,B 0,C 180,E1 -8034.139,E2 -8034.139} C_VEL
LIN {X 0,Y 469.18,Z 747.461,A -85,B 0,C 180,E1 -8034.857,E2 -8034.857} C_VEL
LIN {X 0,Y 470.042,Z 735.484,A -85,B 0,C 180,E1 -8035.458,E2 -8035.458} C_VEL
LIN {X 0,Y 470.812,Z 721.916,A -85,B 0,C 180,E1 -8036.021,E2 -8036.021} C_VEL
LIN {X 0,Y 471.473,Z 709.096,A -85,B 0,C 180,E1 -8036.438,E2 -8036.438} C_VEL
LIN {X 0,Y 471.983,Z 695.299,A -85,B 0,C 180,E1 -8036.774,E2 -8036.774} C_VEL
LIN {X 0,Y 472.745,Z 652.774,A -85,B 0,C 180,E1 -8037.472,E2 -8037.472} C_VEL
LIN {X 0,Y 474.829,Z 513.177,A -85,B 0,C 180,E1 -8039.692,E2 -8039.692} C_VEL
LIN {X 0,Y 467.041,Z 482.37,A -85,B 0,C 180,E1 -8040.78,E2 -8040.78} C_VEL
LIN {X 0,Y 467.063,Z 480.492,A -85,B 0,C 180,E1 -8041.023,E2 -8041.023} C_VEL
LIN {X 0,Y 467.271,Z 477.489,A -85,B 0,C 180,E1 -8041.51,E2 -8041.51} C_VEL
LIN {X 0,Y 465.35,Z 468.706,A -85,B 0,C 180,E1 -8043.132,E2 -8043.132} C_VEL
LIN {X 0,Y 462.19,Z 456.45,A -85,B 0,C 180,E1 -8045.503,E2 -8045.503} C_VEL
LIN {X 0,Y 460.544,Z 450.566,A -85,B 0,C 180,E1 -8046.726,E2 -8046.726} C_VEL
LIN {X 0,Y 460.53,Z 450.337,A -85,B 0,C 180,E1 -8048.895,E2 -8048.895} C_VEL
LIN {X 0,Y 460.517,Z 450.362,A -85,B 0,C 180,E1 -8052.181,E2 -8052.181} C_VEL
LIN {X 0,Y 460.516,Z 450.362,A -85,B 0,C 180,E1 -8055.411,E2 -8055.411} C_VEL
LIN {X 0,Y 460.537,Z 450.365,A -85,B 0,C 180,E1 -8058.395,E2 -8058.395} C_VEL
LIN {X 0,Y 460.537,Z 450.361,A -85,B 0,C 180,E1 -8061.268,E2 -8061.268} C_VEL
LIN {X 0,Y 460.506,Z 450.353,A -85,B 0,C 180,E1 -8064.554,E2 -8064.554} C_VEL
LIN {X 0,Y 460.525,Z 450.37,A -85,B 0,C 180,E1 -8067.715,E2 -8067.715} C_VEL
LIN {X 0,Y 460.538,Z 450.344,A -85,B 0,C 180,E1 -8070.769,E2 -8070.769} C_VEL
LIN {X 0,Y 460.56,Z 450.352,A -85,B 0,C 180,E1 -8073.735,E2 -8073.735} C_VEL
LIN {X 0,Y 460.538,Z 450.362,A -85,B 0,C 180,E1 -8076.624,E2 -8076.624} C_VEL
LIN {X 0,Y 460.542,Z 450.333,A -85,B 0,C 180,E1 -8079.452,E2 -8079.452} C_VEL
LIN {X 0,Y 460.55,Z 450.352,A -85,B 0,C 180,E1 -8082.23,E2 -8082.23} C_VEL
LIN {X 0,Y 460.556,Z 450.361,A -85,B 0,C 180,E1 -8084.964,E2 -8084.964} C_VEL
LIN {X 0,Y 460.604,Z 450.361,A -85,B 0,C 180,E1 -8088.559,E2 -8088.559} C_VEL
LIN {X 0,Y 460.686,Z 450.34,A -85,B 0,C 180,E1 -8092.108,E2 -8092.108} C_VEL
LIN {X 0,Y 460.69,Z 450.346,A -85,B 0,C 180,E1 -8094.748,E2 -8094.748} C_VEL
LIN {X 0,Y 460.816,Z 450.326,A -85,B 0,C 180,E1 -8097.377,E2 -8097.377} C_VEL
LIN {X 0,Y 460.843,Z 450.328,A -85,B 0,C 180,E1 -8100,E2 -8100} C_VEL
LIN {X 0,Y 460.816,Z 450.329,A -85,B 0,C 180,E1 -8102.622,E2 -8102.622} C_VEL
LIN {X 0,Y 460.705,Z 450.338,A -85,B 0,C 180,E1 -8106.13,E2 -8106.13} C_VEL
LIN {X 0,Y 460.62,Z 450.358,A -85,B 0,C 180,E1 -8108.776,E2 -8108.776} C_VEL
LIN {X 0,Y 460.604,Z 450.354,A -85,B 0,C 180,E1 -8112.445,E2 -8112.445} C_VEL
LIN {X 0,Y 460.59,Z 450.349,A -85,B 0,C 180,E1 -8115.998,E2 -8115.998} C_VEL
LIN {X 0,Y 460.562,Z 450.364,A -85,B 0,C 180,E1 -8118.902,E2 -8118.902} C_VEL
LIN {X 0,Y 460.507,Z 450.369,A -85,B 0,C 180,E1 -8121.486,E2 -8121.486} C_VEL
LIN {X 0,Y 460.533,Z 450.364,A -85,B 0,C 180,E1 -8124.332,E2 -8124.332} C_VEL
LIN {X 0,Y 460.574,Z 450.335,A -85,B 0,C 180,E1 -8127.243,E2 -8127.243} C_VEL
LIN {X 0,Y 460.518,Z 450.368,A -85,B 0,C 180,E1 -8130.239,E2 -8130.239} C_VEL
LIN {X 0,Y 460.52,Z 450.343,A -85,B 0,C 180,E1 -8133.325,E2 -8133.325} C_VEL
LIN {X 0,Y 460.472,Z 450.372,A -85,B 0,C 180,E1 -8136.529,E2 -8136.529} C_VEL
LIN {X 0,Y 460.571,Z 450.363,A -85,B 0,C 180,E1 -8139.858,E2 -8139.858} C_VEL
LIN {X 0,Y 460.535,Z 450.37,A -85,B 0,C 180,E1 -8142.905,E2 -8142.905} C_VEL
LIN {X 0,Y 460.504,Z 450.373,A -85,B 0,C 180,E1 -8145.831,E2 -8145.831} C_VEL
LIN {X 0,Y 460.532,Z 450.37,A -85,B 0,C 180,E1 -8148.99,E2 -8148.99} C_VEL
LIN {X 0,Y 460.537,Z 450.371,A -85,B 0,C 180,E1 -8151.269,E2 -8151.269} C_VEL
LIN {X 0,Y 460.507,Z 450.369,A -85,B 0,C 180,E1 -8154.555,E2 -8154.555} C_VEL
LIN {X 0,Y 460.526,Z 450.373,A -85,B 0,C 180,E1 -8157.716,E2 -8157.716} C_VEL
LIN {X 0,Y 460.534,Z 450.368,A -85,B 0,C 180,E1 -8160.769,E2 -8160.769} C_VEL
LIN {X 0,Y 460.563,Z 450.367,A -85,B 0,C 180,E1 -8163.735,E2 -8163.735} C_VEL
LIN {X 0,Y 460.542,Z 450.367,A -85,B 0,C 180,E1 -8166.624,E2 -8166.624} C_VEL
LIN {X 0,Y 460.547,Z 450.371,A -85,B 0,C 180,E1 -8169.453,E2 -8169.453} C_VEL
LIN {X 0,Y 460.555,Z 450.366,A -85,B 0,C 180,E1 -8172.23,E2 -8172.23} C_VEL
LIN {X 0,Y 460.562,Z 450.366,A -85,B 0,C 180,E1 -8174.965,E2 -8174.965} C_VEL
LIN {X 0,Y 460.626,Z 450.361,A -85,B 0,C 180,E1 -8177.667,E2 -8177.667} C_VEL
LIN {X 0,Y 460.583,Z 450.363,A -85,B 0,C 180,E1 -8179.236,E2 -8179.236} C_VEL
LIN {X 0,Y 459.922,Z 450.448,A -85,B 0,C 180,E1 -8179.966,E2 -8179.966} C_VEL
LIN {X 0,Y 457.1,Z 450.801,A -85,B 0,C 180,E1 -8181.153,E2 -8181.153} C_VEL
LIN {X 0,Y 454.721,Z 451.095,A -85,B 0,C 180,E1 -8182.11,E2 -8182.11} C_VEL
LIN {X 0,Y 453.71,Z 451.219,A -85,B 0,C 180,E1 -8182.849,E2 -8182.849} C_VEL
LIN {X 0,Y 453.633,Z 451.228,A -85,B 0,C 180,E1 -8183.099,E2 -8183.099} C_VEL
LIN {X 0,Y 453.667,Z 451.224,A -85,B 0,C 180,E1 -8184.667,E2 -8184.667} C_VEL
LIN {X 0,Y 453.762,Z 451.214,A -85,B 0,C 180,E1 -8187.337,E2 -8187.337} C_VEL
LIN {X 0,Y 453.821,Z 451.209,A -85,B 0,C 180,E1 -8190,E2 -8190} C_VEL
LIN {X 0,Y 453.762,Z 451.214,A -85,B 0,C 180,E1 -8192.663,E2 -8192.663} C_VEL
LIN {X 0,Y 453.673,Z 451.224,A -85,B 0,C 180,E1 -8196.225,E2 -8196.225} C_VEL
LIN {X 0,Y 453.589,Z 451.233,A -85,B 0,C 180,E1 -8198.913,E2 -8198.913} C_VEL
LIN {X 0,Y 453.598,Z 451.234,A -85,B 0,C 180,E1 -8202.551,E2 -8202.551} C_VEL
LIN {X 0,Y 453.541,Z 451.241,A -85,B 0,C 180,E1 -8206.196,E2 -8206.196} C_VEL
LIN {X 0,Y 453.516,Z 451.244,A -85,B 0,C 180,E1 -8209.04,E2 -8209.04} C_VEL
LIN {X 0,Y 453.472,Z 451.248,A -85,B 0,C 180,E1 -8211.836,E2 -8211.836} C_VEL
LIN {X 0,Y 453.509,Z 451.247,A -85,B 0,C 180,E1 -8214.734,E2 -8214.734} C_VEL
LIN {X 0,Y 453.532,Z 451.242,A -85,B 0,C 180,E1 -8217.961,E2 -8217.961} C_VEL
LIN {X 0,Y 453.461,Z 451.248,A -85,B 0,C 180,E1 -8221.525,E2 -8221.525} C_VEL
LIN {X 0,Y 453.483,Z 451.25,A -85,B 0,C 180,E1 -8224.777,E2 -8224.777} C_VEL
LIN {X 0,Y 453.477,Z 451.25,A -85,B 0,C 180,E1 -8228.309,E2 -8228.309} C_VEL
LIN {X 0,Y 453.509,Z 451.247,A -85,B 0,C 180,E1 -8230.606,E2 -8230.606} C_VEL
LIN {X 0,Y 453.458,Z 451.251,A -85,B 0,C 180,E1 -8234.221,E2 -8234.221} C_VEL
LIN {X 0,Y 453.485,Z 451.249,A -85,B 0,C 180,E1 -8237.008,E2 -8237.008} C_VEL
LIN {X 0,Y 453.525,Z 451.244,A -85,B 0,C 180,E1 -8240.555,E2 -8240.555} C_VEL
LIN {X 0,Y 453.449,Z 451.245,A -85,B 0,C 180,E1 -8243.917,E2 -8243.917} C_VEL
LIN {X 0,Y 453.474,Z 451.227,A -85,B 0,C 180,E1 -8247.151,E2 -8247.151} C_VEL
LIN {X 0,Y 453.505,Z 451.242,A -85,B 0,C 180,E1 -8250.271,E2 -8250.271} C_VEL
LIN {X 0,Y 453.504,Z 451.211,A -85,B 0,C 180,E1 -8253.294,E2 -8253.294} C_VEL
LIN {X 0,Y 453.494,Z 451.239,A -85,B 0,C 180,E1 -8256.239,E2 -8256.239} C_VEL
LIN {X 0,Y 453.473,Z 451.243,A -85,B 0,C 180,E1 -8259.118,E2 -8259.118} C_VEL
LIN {X 0,Y 453.502,Z 451.242,A -85,B 0,C 180,E1 -8261.945,E2 -8261.945} C_VEL
LIN {X 0,Y 453.531,Z 451.229,A -85,B 0,C 180,E1 -8264.726,E2 -8264.726} C_VEL
LIN {X 0,Y 453.552,Z 451.227,A -85,B 0,C 180,E1 -8268.379,E2 -8268.379} C_VEL
LIN {X 0,Y 453.643,Z 451.221,A -85,B 0,C 180,E1 -8271.985,E2 -8271.985} C_VEL
LIN {X 0,Y 453.667,Z 451.215,A -85,B 0,C 180,E1 -8274.667,E2 -8274.667} C_VEL
LIN {X 0,Y 453.757,Z 451.21,A -85,B 0,C 180,E1 -8277.337,E2 -8277.337} C_VEL
LIN {X 0,Y 453.814,Z 451.204,A -85,B 0,C 180,E1 -8280,E2 -8280} C_VEL
LIN {X 0,Y 453.757,Z 451.206,A -85,B 0,C 180,E1 -8282.663,E2 -8282.663} C_VEL
LIN {X 0,Y 453.668,Z 451.221,A -85,B 0,C 180,E1 -8286.226,E2 -8286.226} C_VEL
LIN {X 0,Y 453.584,Z 451.22,A -85,B 0,C 180,E1 -8288.914,E2 -8288.914} C_VEL
LIN {X 0,Y 453.555,Z 451.228,A -85,B 0,C 180,E1 -8292.529,E2 -8292.529} C_VEL
LIN {X 0,Y 453.536,Z 451.237,A -85,B 0,C 180,E1 -8296.196,E2 -8296.196} C_VEL
LIN {X 0,Y 453.511,Z 451.215,A -85,B 0,C 180,E1 -8299.041,E2 -8299.041} C_VEL
LIN {X 0,Y 453.468,Z 451.227,A -85,B 0,C 180,E1 -8301.837,E2 -8301.837} C_VEL
LIN {X 0,Y 453.506,Z 451.241,A -85,B 0,C 180,E1 -8304.735,E2 -8304.735} C_VEL
LIN {X 0,Y 453.531,Z 451.21,A -85,B 0,C 180,E1 -8307.962,E2 -8307.962} C_VEL
LIN {X 0,Y 453.476,Z 451.244,A -85,B 0,C 180,E1 -8310.76,E2 -8310.76} C_VEL
LIN {X 0,Y 453.471,Z 451.235,A -85,B 0,C 180,E1 -8313.913,E2 -8313.913} C_VEL
LIN {X 0,Y 453.465,Z 451.247,A -85,B 0,C 180,E1 -8317.188,E2 -8317.188} C_VEL
LIN {X 0,Y 453.525,Z 451.231,A -85,B 0,C 180,E1 -8319.446,E2 -8319.446} C_VEL
LIN {X 0,Y 453.486,Z 451.242,A -85,B 0,C 180,E1 -8322.992,E2 -8322.992} C_VEL
LIN {X 0,Y 453.461,Z 451.249,A -85,B 0,C 180,E1 -8325.78,E2 -8325.78} C_VEL
LIN {X 0,Y 453.474,Z 451.24,A -85,B 0,C 180,E1 -8328.21,E2 -8328.21} C_VEL
LIN {X 0,Y 453.467,Z 451.22,A -85,B 0,C 180,E1 -8330.797,E2 -8330.797} C_VEL
LIN {X 0,Y 453.504,Z 451.434,A -85,B 0,C 180,E1 -8332.816,E2 -8332.816} C_VEL
LIN {X 0,Y 457.401,Z 465.83,A -85,B 0,C 180,E1 -8335.769,E2 -8335.769} C_VEL
LIN {X 0,Y 460.223,Z 477.209,A -85,B 0,C 180,E1 -8337.951,E2 -8337.951} C_VEL
LIN {X 0,Y 460.427,Z 481.118,A -85,B 0,C 180,E1 -8338.622,E2 -8338.622} C_VEL
LIN {X 0,Y 460.534,Z 482.496,A -85,B 0,C 180,E1 -8338.745,E2 -8338.745} C_VEL
LIN {X 0,Y 468.609,Z 514.574,A -85,B 0,C 180,E1 -8339.902,E2 -8339.902} C_VEL
LIN {X 0,Y 466.451,Z 652.564,A -85,B 0,C 180,E1 -8342.126,E2 -8342.126} C_VEL
LIN {X 0,Y 465.631,Z 694.568,A -85,B 0,C 180,E1 -8342.82,E2 -8342.82} C_VEL
LIN {X 0,Y 465.099,Z 708.27,A -85,B 0,C 180,E1 -8343.153,E2 -8343.153} C_VEL
LIN {X 0,Y 464.428,Z 721.731,A -85,B 0,C 180,E1 -8343.595,E2 -8343.595} C_VEL
LIN {X 0,Y 463.555,Z 735.271,A -85,B 0,C 180,E1 -8344.159,E2 -8344.159} C_VEL
LIN {X 0,Y 462.503,Z 750.33,A -85,B 0,C 180,E1 -8344.94,E2 -8344.94} C_VEL
LIN {X 0,Y 461.234,Z 766.199,A -85,B 0,C 180,E1 -8345.967,E2 -8345.967} C_VEL
LIN {X 0,Y 460.067,Z 778.968,A -85,B 0,C 180,E1 -8346.956,E2 -8346.956} C_VEL
LIN {X 0,Y 458.958,Z 790.271,A -85,B 0,C 180,E1 -8347.966,E2 -8347.966} C_VEL
LIN {X 0,Y 457.921,Z 801.257,A -85,B 0,C 180,E1 -8349.095,E2 -8349.095} C_VEL
LIN {X 0,Y 456.977,Z 810.954,A -85,B 0,C 180,E1 -8350.224,E2 -8350.224} C_VEL
LIN {X 0,Y 455.966,Z 821.166,A -85,B 0,C 180,E1 -8351.581,E2 -8351.581} C_VEL
LIN {X 0,Y 455.187,Z 830.13,A -85,B 0,C 180,E1 -8352.941,E2 -8352.941} C_VEL
LIN {X 0,Y 454.545,Z 838.025,A -85,B 0,C 180,E1 -8354.302,E2 -8354.302} C_VEL
LIN {X 0,Y 453.938,Z 844.986,A -85,B 0,C 180,E1 -8355.658,E2 -8355.658} C_VEL
LIN {X 0,Y 453.54,Z 851.126,A -85,B 0,C 180,E1 -8357.016,E2 -8357.016} C_VEL
LIN {X 0,Y 453.081,Z 858.066,A -85,B 0,C 180,E1 -8358.82,E2 -8358.82} C_VEL
LIN {X 0,Y 452.759,Z 863.813,A -85,B 0,C 180,E1 -8360.62,E2 -8360.62} C_VEL
LIN {X 0,Y 452.636,Z 867.418,A -85,B 0,C 180,E1 -8361.967,E2 -8361.967} C_VEL
LIN {X 0,Y 452.561,Z 871.258,A -85,B 0,C 180,E1 -8363.759,E2 -8363.759} C_VEL
LIN {X 0,Y 452.44,Z 874.094,A -85,B 0,C 180,E1 -8365.546,E2 -8365.546} C_VEL
LIN {X 0,Y 452.481,Z 875.969,A -85,B 0,C 180,E1 -8367.329,E2 -8367.329} C_VEL
LIN {X 0,Y 452.426,Z 876.64,A -85,B 0,C 180,E1 -8368.22,E2 -8368.22} C_VEL
LIN {X 0,Y 452.376,Z 877.108,A -85,B 0,C 180,E1 -8370,E2 -8370} C_VEL
LIN {X 0,Y 452.426,Z 876.64,A -85,B 0,C 180,E1 -8371.78,E2 -8371.78} C_VEL
LIN {X 0,Y 452.432,Z 875.224,A -85,B 0,C 180,E1 -8373.562,E2 -8373.562} C_VEL
LIN {X 0,Y 452.499,Z 872.852,A -85,B 0,C 180,E1 -8375.347,E2 -8375.347} C_VEL
LIN {X 0,Y 452.642,Z 869.493,A -85,B 0,C 180,E1 -8377.135,E2 -8377.135} C_VEL
LIN {X 0,Y 452.715,Z 865.097,A -85,B 0,C 180,E1 -8378.931,E2 -8378.931} C_VEL
LIN {X 0,Y 452.972,Z 859.607,A -85,B 0,C 180,E1 -8380.73,E2 -8380.73} C_VEL
LIN {X 0,Y 453.248,Z 855.036,A -85,B 0,C 180,E1 -8382.012,E2 -8382.012} C_VEL
LIN {X 0,Y 453.801,Z 847.092,A -85,B 0,C 180,E1 -8383.889,E2 -8383.889} C_VEL
LIN {X 0,Y 454.301,Z 840.441,A -85,B 0,C 180,E1 -8385.247,E2 -8385.247} C_VEL
LIN {X 0,Y 454.962,Z 833.053,A -85,B 0,C 180,E1 -8386.578,E2 -8386.578} C_VEL
LIN {X 0,Y 455.682,Z 824.3,A -85,B 0,C 180,E1 -8387.966,E2 -8387.966} C_VEL
LIN {X 0,Y 456.604,Z 814.506,A -85,B 0,C 180,E1 -8389.324,E2 -8389.324} C_VEL
LIN {X 0,Y 457.61,Z 804.427,A -85,B 0,C 180,E1 -8390.55,E2 -8390.55} C_VEL
LIN {X 0,Y 458.641,Z 793.705,A -85,B 0,C 180,E1 -8391.695,E2 -8391.695} C_VEL
LIN {X 0,Y 459.641,Z 782.885,A -85,B 0,C 180,E1 -8392.71,E2 -8392.71} C_VEL
